;FOLD LIN P2869 Vel=2 m/s CPDAT2869 Tool[1]:marker Base[0] ;%{PE}
;FOLD Parameters ;%{h}
;Params IlfProvider=kukaroboter.basistech.inlineforms.movement.old; Kuka.IsGlobalPoint=False; Kuka.PointName=P2869; Kuka.BlendingEnabled=False; Kuka.MoveDataName=CPDAT1; Kuka.VelocityPath=2; Kuka.CurrentCDSetIndex=0; Kuka.MovementParameterFieldEnabled=True; IlfCommand=LIN
;ENDFOLD
$BWDSTART = FALSE
LDAT_ACT = LCPDAT2869
FDAT_ACT = FP2869
BAS(#CP_PARAMS, 2.0)
SET_CD_PARAMS (0)
LIN XP2869
;ENDFOLD

;FOLD LIN P2870 Vel=2 m/s CPDAT2870 Tool[1]:marker Base[0] ;%{PE}
;FOLD Parameters ;%{h}
;Params IlfProvider=kukaroboter.basistech.inlineforms.movement.old; Kuka.IsGlobalPoint=False; Kuka.PointName=P2870; Kuka.BlendingEnabled=False; Kuka.MoveDataName=CPDAT1; Kuka.VelocityPath=2; Kuka.CurrentCDSetIndex=0; Kuka.MovementParameterFieldEnabled=True; IlfCommand=LIN
;ENDFOLD
$BWDSTART = FALSE
LDAT_ACT = LCPDAT2870
FDAT_ACT = FP2870
BAS(#CP_PARAMS, 2.0)
SET_CD_PARAMS (0)
LIN XP2870
;ENDFOLD

;FOLD LIN P2871 Vel=2 m/s CPDAT2871 Tool[1]:marker Base[0] ;%{PE}
;FOLD Parameters ;%{h}
;Params IlfProvider=kukaroboter.basistech.inlineforms.movement.old; Kuka.IsGlobalPoint=False; Kuka.PointName=P2871; Kuka.BlendingEnabled=False; Kuka.MoveDataName=CPDAT1; Kuka.VelocityPath=2; Kuka.CurrentCDSetIndex=0; Kuka.MovementParameterFieldEnabled=True; IlfCommand=LIN
;ENDFOLD
$BWDSTART = FALSE
LDAT_ACT = LCPDAT2871
FDAT_ACT = FP2871
BAS(#CP_PARAMS, 2.0)
SET_CD_PARAMS (0)
LIN XP2871
;ENDFOLD

;FOLD LIN P2872 Vel=2 m/s CPDAT2872 Tool[1]:marker Base[0] ;%{PE}
;FOLD Parameters ;%{h}
;Params IlfProvider=kukaroboter.basistech.inlineforms.movement.old; Kuka.IsGlobalPoint=False; Kuka.PointName=P2872; Kuka.BlendingEnabled=False; Kuka.MoveDataName=CPDAT1; Kuka.VelocityPath=2; Kuka.CurrentCDSetIndex=0; Kuka.MovementParameterFieldEnabled=True; IlfCommand=LIN
;ENDFOLD
$BWDSTART = FALSE
LDAT_ACT = LCPDAT2872
FDAT_ACT = FP2872
BAS(#CP_PARAMS, 2.0)
SET_CD_PARAMS (0)
LIN XP2872
;ENDFOLD

;FOLD LIN P2873 Vel=2 m/s CPDAT2873 Tool[1]:marker Base[0] ;%{PE}
;FOLD Parameters ;%{h}
;Params IlfProvider=kukaroboter.basistech.inlineforms.movement.old; Kuka.IsGlobalPoint=False; Kuka.PointName=P2873; Kuka.BlendingEnabled=False; Kuka.MoveDataName=CPDAT1; Kuka.VelocityPath=2; Kuka.CurrentCDSetIndex=0; Kuka.MovementParameterFieldEnabled=True; IlfCommand=LIN
;ENDFOLD
$BWDSTART = FALSE
LDAT_ACT = LCPDAT2873
FDAT_ACT = FP2873
BAS(#CP_PARAMS, 2.0)
SET_CD_PARAMS (0)
LIN XP2873
;ENDFOLD

;FOLD LIN P2874 Vel=2 m/s CPDAT2874 Tool[1]:marker Base[0] ;%{PE}
;FOLD Parameters ;%{h}
;Params IlfProvider=kukaroboter.basistech.inlineforms.movement.old; Kuka.IsGlobalPoint=False; Kuka.PointName=P2874; Kuka.BlendingEnabled=False; Kuka.MoveDataName=CPDAT1; Kuka.VelocityPath=2; Kuka.CurrentCDSetIndex=0; Kuka.MovementParameterFieldEnabled=True; IlfCommand=LIN
;ENDFOLD
$BWDSTART = FALSE
LDAT_ACT = LCPDAT2874
FDAT_ACT = FP2874
BAS(#CP_PARAMS, 2.0)
SET_CD_PARAMS (0)
LIN XP2874
;ENDFOLD

;FOLD LIN P2875 Vel=2 m/s CPDAT2875 Tool[1]:marker Base[0] ;%{PE}
;FOLD Parameters ;%{h}
;Params IlfProvider=kukaroboter.basistech.inlineforms.movement.old; Kuka.IsGlobalPoint=False; Kuka.PointName=P2875; Kuka.BlendingEnabled=False; Kuka.MoveDataName=CPDAT1; Kuka.VelocityPath=2; Kuka.CurrentCDSetIndex=0; Kuka.MovementParameterFieldEnabled=True; IlfCommand=LIN
;ENDFOLD
$BWDSTART = FALSE
LDAT_ACT = LCPDAT2875
FDAT_ACT = FP2875
BAS(#CP_PARAMS, 2.0)
SET_CD_PARAMS (0)
LIN XP2875
;ENDFOLD

;FOLD LIN P2876 Vel=2 m/s CPDAT2876 Tool[1]:marker Base[0] ;%{PE}
;FOLD Parameters ;%{h}
;Params IlfProvider=kukaroboter.basistech.inlineforms.movement.old; Kuka.IsGlobalPoint=False; Kuka.PointName=P2876; Kuka.BlendingEnabled=False; Kuka.MoveDataName=CPDAT1; Kuka.VelocityPath=2; Kuka.CurrentCDSetIndex=0; Kuka.MovementParameterFieldEnabled=True; IlfCommand=LIN
;ENDFOLD
$BWDSTART = FALSE
LDAT_ACT = LCPDAT2876
FDAT_ACT = FP2876
BAS(#CP_PARAMS, 2.0)
SET_CD_PARAMS (0)
LIN XP2876
;ENDFOLD

;FOLD LIN P2877 Vel=2 m/s CPDAT2877 Tool[1]:marker Base[0] ;%{PE}
;FOLD Parameters ;%{h}
;Params IlfProvider=kukaroboter.basistech.inlineforms.movement.old; Kuka.IsGlobalPoint=False; Kuka.PointName=P2877; Kuka.BlendingEnabled=False; Kuka.MoveDataName=CPDAT1; Kuka.VelocityPath=2; Kuka.CurrentCDSetIndex=0; Kuka.MovementParameterFieldEnabled=True; IlfCommand=LIN
;ENDFOLD
$BWDSTART = FALSE
LDAT_ACT = LCPDAT2877
FDAT_ACT = FP2877
BAS(#CP_PARAMS, 2.0)
SET_CD_PARAMS (0)
LIN XP2877
;ENDFOLD

;FOLD LIN P2878 Vel=2 m/s CPDAT2878 Tool[1]:marker Base[0] ;%{PE}
;FOLD Parameters ;%{h}
;Params IlfProvider=kukaroboter.basistech.inlineforms.movement.old; Kuka.IsGlobalPoint=False; Kuka.PointName=P2878; Kuka.BlendingEnabled=False; Kuka.MoveDataName=CPDAT1; Kuka.VelocityPath=2; Kuka.CurrentCDSetIndex=0; Kuka.MovementParameterFieldEnabled=True; IlfCommand=LIN
;ENDFOLD
$BWDSTART = FALSE
LDAT_ACT = LCPDAT2878
FDAT_ACT = FP2878
BAS(#CP_PARAMS, 2.0)
SET_CD_PARAMS (0)
LIN XP2878
;ENDFOLD

;FOLD LIN P2879 Vel=2 m/s CPDAT2879 Tool[1]:marker Base[0] ;%{PE}
;FOLD Parameters ;%{h}
;Params IlfProvider=kukaroboter.basistech.inlineforms.movement.old; Kuka.IsGlobalPoint=False; Kuka.PointName=P2879; Kuka.BlendingEnabled=False; Kuka.MoveDataName=CPDAT1; Kuka.VelocityPath=2; Kuka.CurrentCDSetIndex=0; Kuka.MovementParameterFieldEnabled=True; IlfCommand=LIN
;ENDFOLD
$BWDSTART = FALSE
LDAT_ACT = LCPDAT2879
FDAT_ACT = FP2879
BAS(#CP_PARAMS, 2.0)
SET_CD_PARAMS (0)
LIN XP2879
;ENDFOLD

;FOLD LIN P2880 Vel=2 m/s CPDAT2880 Tool[1]:marker Base[0] ;%{PE}
;FOLD Parameters ;%{h}
;Params IlfProvider=kukaroboter.basistech.inlineforms.movement.old; Kuka.IsGlobalPoint=False; Kuka.PointName=P2880; Kuka.BlendingEnabled=False; Kuka.MoveDataName=CPDAT1; Kuka.VelocityPath=2; Kuka.CurrentCDSetIndex=0; Kuka.MovementParameterFieldEnabled=True; IlfCommand=LIN
;ENDFOLD
$BWDSTART = FALSE
LDAT_ACT = LCPDAT2880
FDAT_ACT = FP2880
BAS(#CP_PARAMS, 2.0)
SET_CD_PARAMS (0)
LIN XP2880
;ENDFOLD

;FOLD LIN P2881 Vel=2 m/s CPDAT2881 Tool[1]:marker Base[0] ;%{PE}
;FOLD Parameters ;%{h}
;Params IlfProvider=kukaroboter.basistech.inlineforms.movement.old; Kuka.IsGlobalPoint=False; Kuka.PointName=P2881; Kuka.BlendingEnabled=False; Kuka.MoveDataName=CPDAT1; Kuka.VelocityPath=2; Kuka.CurrentCDSetIndex=0; Kuka.MovementParameterFieldEnabled=True; IlfCommand=LIN
;ENDFOLD
$BWDSTART = FALSE
LDAT_ACT = LCPDAT2881
FDAT_ACT = FP2881
BAS(#CP_PARAMS, 2.0)
SET_CD_PARAMS (0)
LIN XP2881
;ENDFOLD

;FOLD LIN P2882 Vel=2 m/s CPDAT2882 Tool[1]:marker Base[0] ;%{PE}
;FOLD Parameters ;%{h}
;Params IlfProvider=kukaroboter.basistech.inlineforms.movement.old; Kuka.IsGlobalPoint=False; Kuka.PointName=P2882; Kuka.BlendingEnabled=False; Kuka.MoveDataName=CPDAT1; Kuka.VelocityPath=2; Kuka.CurrentCDSetIndex=0; Kuka.MovementParameterFieldEnabled=True; IlfCommand=LIN
;ENDFOLD
$BWDSTART = FALSE
LDAT_ACT = LCPDAT2882
FDAT_ACT = FP2882
BAS(#CP_PARAMS, 2.0)
SET_CD_PARAMS (0)
LIN XP2882
;ENDFOLD

;FOLD LIN P2883 Vel=2 m/s CPDAT2883 Tool[1]:marker Base[0] ;%{PE}
;FOLD Parameters ;%{h}
;Params IlfProvider=kukaroboter.basistech.inlineforms.movement.old; Kuka.IsGlobalPoint=False; Kuka.PointName=P2883; Kuka.BlendingEnabled=False; Kuka.MoveDataName=CPDAT1; Kuka.VelocityPath=2; Kuka.CurrentCDSetIndex=0; Kuka.MovementParameterFieldEnabled=True; IlfCommand=LIN
;ENDFOLD
$BWDSTART = FALSE
LDAT_ACT = LCPDAT2883
FDAT_ACT = FP2883
BAS(#CP_PARAMS, 2.0)
SET_CD_PARAMS (0)
LIN XP2883
;ENDFOLD

;FOLD LIN P2884 Vel=2 m/s CPDAT2884 Tool[1]:marker Base[0] ;%{PE}
;FOLD Parameters ;%{h}
;Params IlfProvider=kukaroboter.basistech.inlineforms.movement.old; Kuka.IsGlobalPoint=False; Kuka.PointName=P2884; Kuka.BlendingEnabled=False; Kuka.MoveDataName=CPDAT1; Kuka.VelocityPath=2; Kuka.CurrentCDSetIndex=0; Kuka.MovementParameterFieldEnabled=True; IlfCommand=LIN
;ENDFOLD
$BWDSTART = FALSE
LDAT_ACT = LCPDAT2884
FDAT_ACT = FP2884
BAS(#CP_PARAMS, 2.0)
SET_CD_PARAMS (0)
LIN XP2884
;ENDFOLD

;FOLD LIN P2885 Vel=2 m/s CPDAT2885 Tool[1]:marker Base[0] ;%{PE}
;FOLD Parameters ;%{h}
;Params IlfProvider=kukaroboter.basistech.inlineforms.movement.old; Kuka.IsGlobalPoint=False; Kuka.PointName=P2885; Kuka.BlendingEnabled=False; Kuka.MoveDataName=CPDAT1; Kuka.VelocityPath=2; Kuka.CurrentCDSetIndex=0; Kuka.MovementParameterFieldEnabled=True; IlfCommand=LIN
;ENDFOLD
$BWDSTART = FALSE
LDAT_ACT = LCPDAT2885
FDAT_ACT = FP2885
BAS(#CP_PARAMS, 2.0)
SET_CD_PARAMS (0)
LIN XP2885
;ENDFOLD

;FOLD LIN P2886 Vel=2 m/s CPDAT2886 Tool[1]:marker Base[0] ;%{PE}
;FOLD Parameters ;%{h}
;Params IlfProvider=kukaroboter.basistech.inlineforms.movement.old; Kuka.IsGlobalPoint=False; Kuka.PointName=P2886; Kuka.BlendingEnabled=False; Kuka.MoveDataName=CPDAT1; Kuka.VelocityPath=2; Kuka.CurrentCDSetIndex=0; Kuka.MovementParameterFieldEnabled=True; IlfCommand=LIN
;ENDFOLD
$BWDSTART = FALSE
LDAT_ACT = LCPDAT2886
FDAT_ACT = FP2886
BAS(#CP_PARAMS, 2.0)
SET_CD_PARAMS (0)
LIN XP2886
;ENDFOLD

;FOLD LIN P2887 Vel=2 m/s CPDAT2887 Tool[1]:marker Base[0] ;%{PE}
;FOLD Parameters ;%{h}
;Params IlfProvider=kukaroboter.basistech.inlineforms.movement.old; Kuka.IsGlobalPoint=False; Kuka.PointName=P2887; Kuka.BlendingEnabled=False; Kuka.MoveDataName=CPDAT1; Kuka.VelocityPath=2; Kuka.CurrentCDSetIndex=0; Kuka.MovementParameterFieldEnabled=True; IlfCommand=LIN
;ENDFOLD
$BWDSTART = FALSE
LDAT_ACT = LCPDAT2887
FDAT_ACT = FP2887
BAS(#CP_PARAMS, 2.0)
SET_CD_PARAMS (0)
LIN XP2887
;ENDFOLD

;FOLD LIN P2888 Vel=2 m/s CPDAT2888 Tool[1]:marker Base[0] ;%{PE}
;FOLD Parameters ;%{h}
;Params IlfProvider=kukaroboter.basistech.inlineforms.movement.old; Kuka.IsGlobalPoint=False; Kuka.PointName=P2888; Kuka.BlendingEnabled=False; Kuka.MoveDataName=CPDAT1; Kuka.VelocityPath=2; Kuka.CurrentCDSetIndex=0; Kuka.MovementParameterFieldEnabled=True; IlfCommand=LIN
;ENDFOLD
$BWDSTART = FALSE
LDAT_ACT = LCPDAT2888
FDAT_ACT = FP2888
BAS(#CP_PARAMS, 2.0)
SET_CD_PARAMS (0)
LIN XP2888
;ENDFOLD

;FOLD LIN P2889 Vel=2 m/s CPDAT2889 Tool[1]:marker Base[0] ;%{PE}
;FOLD Parameters ;%{h}
;Params IlfProvider=kukaroboter.basistech.inlineforms.movement.old; Kuka.IsGlobalPoint=False; Kuka.PointName=P2889; Kuka.BlendingEnabled=False; Kuka.MoveDataName=CPDAT1; Kuka.VelocityPath=2; Kuka.CurrentCDSetIndex=0; Kuka.MovementParameterFieldEnabled=True; IlfCommand=LIN
;ENDFOLD
$BWDSTART = FALSE
LDAT_ACT = LCPDAT2889
FDAT_ACT = FP2889
BAS(#CP_PARAMS, 2.0)
SET_CD_PARAMS (0)
LIN XP2889
;ENDFOLD

;FOLD LIN P2890 Vel=2 m/s CPDAT2890 Tool[1]:marker Base[0] ;%{PE}
;FOLD Parameters ;%{h}
;Params IlfProvider=kukaroboter.basistech.inlineforms.movement.old; Kuka.IsGlobalPoint=False; Kuka.PointName=P2890; Kuka.BlendingEnabled=False; Kuka.MoveDataName=CPDAT1; Kuka.VelocityPath=2; Kuka.CurrentCDSetIndex=0; Kuka.MovementParameterFieldEnabled=True; IlfCommand=LIN
;ENDFOLD
$BWDSTART = FALSE
LDAT_ACT = LCPDAT2890
FDAT_ACT = FP2890
BAS(#CP_PARAMS, 2.0)
SET_CD_PARAMS (0)
LIN XP2890
;ENDFOLD

;FOLD LIN P2891 Vel=2 m/s CPDAT2891 Tool[1]:marker Base[0] ;%{PE}
;FOLD Parameters ;%{h}
;Params IlfProvider=kukaroboter.basistech.inlineforms.movement.old; Kuka.IsGlobalPoint=False; Kuka.PointName=P2891; Kuka.BlendingEnabled=False; Kuka.MoveDataName=CPDAT1; Kuka.VelocityPath=2; Kuka.CurrentCDSetIndex=0; Kuka.MovementParameterFieldEnabled=True; IlfCommand=LIN
;ENDFOLD
$BWDSTART = FALSE
LDAT_ACT = LCPDAT2891
FDAT_ACT = FP2891
BAS(#CP_PARAMS, 2.0)
SET_CD_PARAMS (0)
LIN XP2891
;ENDFOLD

;FOLD LIN P2892 Vel=2 m/s CPDAT2892 Tool[1]:marker Base[0] ;%{PE}
;FOLD Parameters ;%{h}
;Params IlfProvider=kukaroboter.basistech.inlineforms.movement.old; Kuka.IsGlobalPoint=False; Kuka.PointName=P2892; Kuka.BlendingEnabled=False; Kuka.MoveDataName=CPDAT1; Kuka.VelocityPath=2; Kuka.CurrentCDSetIndex=0; Kuka.MovementParameterFieldEnabled=True; IlfCommand=LIN
;ENDFOLD
$BWDSTART = FALSE
LDAT_ACT = LCPDAT2892
FDAT_ACT = FP2892
BAS(#CP_PARAMS, 2.0)
SET_CD_PARAMS (0)
LIN XP2892
;ENDFOLD

;FOLD LIN P2893 Vel=2 m/s CPDAT2893 Tool[1]:marker Base[0] ;%{PE}
;FOLD Parameters ;%{h}
;Params IlfProvider=kukaroboter.basistech.inlineforms.movement.old; Kuka.IsGlobalPoint=False; Kuka.PointName=P2893; Kuka.BlendingEnabled=False; Kuka.MoveDataName=CPDAT1; Kuka.VelocityPath=2; Kuka.CurrentCDSetIndex=0; Kuka.MovementParameterFieldEnabled=True; IlfCommand=LIN
;ENDFOLD
$BWDSTART = FALSE
LDAT_ACT = LCPDAT2893
FDAT_ACT = FP2893
BAS(#CP_PARAMS, 2.0)
SET_CD_PARAMS (0)
LIN XP2893
;ENDFOLD

;FOLD LIN P2894 Vel=2 m/s CPDAT2894 Tool[1]:marker Base[0] ;%{PE}
;FOLD Parameters ;%{h}
;Params IlfProvider=kukaroboter.basistech.inlineforms.movement.old; Kuka.IsGlobalPoint=False; Kuka.PointName=P2894; Kuka.BlendingEnabled=False; Kuka.MoveDataName=CPDAT1; Kuka.VelocityPath=2; Kuka.CurrentCDSetIndex=0; Kuka.MovementParameterFieldEnabled=True; IlfCommand=LIN
;ENDFOLD
$BWDSTART = FALSE
LDAT_ACT = LCPDAT2894
FDAT_ACT = FP2894
BAS(#CP_PARAMS, 2.0)
SET_CD_PARAMS (0)
LIN XP2894
;ENDFOLD

;FOLD LIN P2895 Vel=2 m/s CPDAT2895 Tool[1]:marker Base[0] ;%{PE}
;FOLD Parameters ;%{h}
;Params IlfProvider=kukaroboter.basistech.inlineforms.movement.old; Kuka.IsGlobalPoint=False; Kuka.PointName=P2895; Kuka.BlendingEnabled=False; Kuka.MoveDataName=CPDAT1; Kuka.VelocityPath=2; Kuka.CurrentCDSetIndex=0; Kuka.MovementParameterFieldEnabled=True; IlfCommand=LIN
;ENDFOLD
$BWDSTART = FALSE
LDAT_ACT = LCPDAT2895
FDAT_ACT = FP2895
BAS(#CP_PARAMS, 2.0)
SET_CD_PARAMS (0)
LIN XP2895
;ENDFOLD

;FOLD LIN P2896 Vel=2 m/s CPDAT2896 Tool[1]:marker Base[0] ;%{PE}
;FOLD Parameters ;%{h}
;Params IlfProvider=kukaroboter.basistech.inlineforms.movement.old; Kuka.IsGlobalPoint=False; Kuka.PointName=P2896; Kuka.BlendingEnabled=False; Kuka.MoveDataName=CPDAT1; Kuka.VelocityPath=2; Kuka.CurrentCDSetIndex=0; Kuka.MovementParameterFieldEnabled=True; IlfCommand=LIN
;ENDFOLD
$BWDSTART = FALSE
LDAT_ACT = LCPDAT2896
FDAT_ACT = FP2896
BAS(#CP_PARAMS, 2.0)
SET_CD_PARAMS (0)
LIN XP2896
;ENDFOLD

;FOLD LIN P2897 Vel=2 m/s CPDAT2897 Tool[1]:marker Base[0] ;%{PE}
;FOLD Parameters ;%{h}
;Params IlfProvider=kukaroboter.basistech.inlineforms.movement.old; Kuka.IsGlobalPoint=False; Kuka.PointName=P2897; Kuka.BlendingEnabled=False; Kuka.MoveDataName=CPDAT1; Kuka.VelocityPath=2; Kuka.CurrentCDSetIndex=0; Kuka.MovementParameterFieldEnabled=True; IlfCommand=LIN
;ENDFOLD
$BWDSTART = FALSE
LDAT_ACT = LCPDAT2897
FDAT_ACT = FP2897
BAS(#CP_PARAMS, 2.0)
SET_CD_PARAMS (0)
LIN XP2897
;ENDFOLD

;FOLD LIN P2898 Vel=2 m/s CPDAT2898 Tool[1]:marker Base[0] ;%{PE}
;FOLD Parameters ;%{h}
;Params IlfProvider=kukaroboter.basistech.inlineforms.movement.old; Kuka.IsGlobalPoint=False; Kuka.PointName=P2898; Kuka.BlendingEnabled=False; Kuka.MoveDataName=CPDAT1; Kuka.VelocityPath=2; Kuka.CurrentCDSetIndex=0; Kuka.MovementParameterFieldEnabled=True; IlfCommand=LIN
;ENDFOLD
$BWDSTART = FALSE
LDAT_ACT = LCPDAT2898
FDAT_ACT = FP2898
BAS(#CP_PARAMS, 2.0)
SET_CD_PARAMS (0)
LIN XP2898
;ENDFOLD

;FOLD LIN P2899 Vel=2 m/s CPDAT2899 Tool[1]:marker Base[0] ;%{PE}
;FOLD Parameters ;%{h}
;Params IlfProvider=kukaroboter.basistech.inlineforms.movement.old; Kuka.IsGlobalPoint=False; Kuka.PointName=P2899; Kuka.BlendingEnabled=False; Kuka.MoveDataName=CPDAT1; Kuka.VelocityPath=2; Kuka.CurrentCDSetIndex=0; Kuka.MovementParameterFieldEnabled=True; IlfCommand=LIN
;ENDFOLD
$BWDSTART = FALSE
LDAT_ACT = LCPDAT2899
FDAT_ACT = FP2899
BAS(#CP_PARAMS, 2.0)
SET_CD_PARAMS (0)
LIN XP2899
;ENDFOLD

;FOLD LIN P2900 Vel=2 m/s CPDAT2900 Tool[1]:marker Base[0] ;%{PE}
;FOLD Parameters ;%{h}
;Params IlfProvider=kukaroboter.basistech.inlineforms.movement.old; Kuka.IsGlobalPoint=False; Kuka.PointName=P2900; Kuka.BlendingEnabled=False; Kuka.MoveDataName=CPDAT1; Kuka.VelocityPath=2; Kuka.CurrentCDSetIndex=0; Kuka.MovementParameterFieldEnabled=True; IlfCommand=LIN
;ENDFOLD
$BWDSTART = FALSE
LDAT_ACT = LCPDAT2900
FDAT_ACT = FP2900
BAS(#CP_PARAMS, 2.0)
SET_CD_PARAMS (0)
LIN XP2900
;ENDFOLD

;FOLD LIN P2901 Vel=2 m/s CPDAT2901 Tool[1]:marker Base[0] ;%{PE}
;FOLD Parameters ;%{h}
;Params IlfProvider=kukaroboter.basistech.inlineforms.movement.old; Kuka.IsGlobalPoint=False; Kuka.PointName=P2901; Kuka.BlendingEnabled=False; Kuka.MoveDataName=CPDAT1; Kuka.VelocityPath=2; Kuka.CurrentCDSetIndex=0; Kuka.MovementParameterFieldEnabled=True; IlfCommand=LIN
;ENDFOLD
$BWDSTART = FALSE
LDAT_ACT = LCPDAT2901
FDAT_ACT = FP2901
BAS(#CP_PARAMS, 2.0)
SET_CD_PARAMS (0)
LIN XP2901
;ENDFOLD

;FOLD LIN P2902 Vel=2 m/s CPDAT2902 Tool[1]:marker Base[0] ;%{PE}
;FOLD Parameters ;%{h}
;Params IlfProvider=kukaroboter.basistech.inlineforms.movement.old; Kuka.IsGlobalPoint=False; Kuka.PointName=P2902; Kuka.BlendingEnabled=False; Kuka.MoveDataName=CPDAT1; Kuka.VelocityPath=2; Kuka.CurrentCDSetIndex=0; Kuka.MovementParameterFieldEnabled=True; IlfCommand=LIN
;ENDFOLD
$BWDSTART = FALSE
LDAT_ACT = LCPDAT2902
FDAT_ACT = FP2902
BAS(#CP_PARAMS, 2.0)
SET_CD_PARAMS (0)
LIN XP2902
;ENDFOLD

;FOLD LIN P2903 Vel=2 m/s CPDAT2903 Tool[1]:marker Base[0] ;%{PE}
;FOLD Parameters ;%{h}
;Params IlfProvider=kukaroboter.basistech.inlineforms.movement.old; Kuka.IsGlobalPoint=False; Kuka.PointName=P2903; Kuka.BlendingEnabled=False; Kuka.MoveDataName=CPDAT1; Kuka.VelocityPath=2; Kuka.CurrentCDSetIndex=0; Kuka.MovementParameterFieldEnabled=True; IlfCommand=LIN
;ENDFOLD
$BWDSTART = FALSE
LDAT_ACT = LCPDAT2903
FDAT_ACT = FP2903
BAS(#CP_PARAMS, 2.0)
SET_CD_PARAMS (0)
LIN XP2903
;ENDFOLD

;FOLD LIN P2904 Vel=2 m/s CPDAT2904 Tool[1]:marker Base[0] ;%{PE}
;FOLD Parameters ;%{h}
;Params IlfProvider=kukaroboter.basistech.inlineforms.movement.old; Kuka.IsGlobalPoint=False; Kuka.PointName=P2904; Kuka.BlendingEnabled=False; Kuka.MoveDataName=CPDAT1; Kuka.VelocityPath=2; Kuka.CurrentCDSetIndex=0; Kuka.MovementParameterFieldEnabled=True; IlfCommand=LIN
;ENDFOLD
$BWDSTART = FALSE
LDAT_ACT = LCPDAT2904
FDAT_ACT = FP2904
BAS(#CP_PARAMS, 2.0)
SET_CD_PARAMS (0)
LIN XP2904
;ENDFOLD

;FOLD LIN P2905 Vel=2 m/s CPDAT2905 Tool[1]:marker Base[0] ;%{PE}
;FOLD Parameters ;%{h}
;Params IlfProvider=kukaroboter.basistech.inlineforms.movement.old; Kuka.IsGlobalPoint=False; Kuka.PointName=P2905; Kuka.BlendingEnabled=False; Kuka.MoveDataName=CPDAT1; Kuka.VelocityPath=2; Kuka.CurrentCDSetIndex=0; Kuka.MovementParameterFieldEnabled=True; IlfCommand=LIN
;ENDFOLD
$BWDSTART = FALSE
LDAT_ACT = LCPDAT2905
FDAT_ACT = FP2905
BAS(#CP_PARAMS, 2.0)
SET_CD_PARAMS (0)
LIN XP2905
;ENDFOLD

;FOLD LIN P2906 Vel=2 m/s CPDAT2906 Tool[1]:marker Base[0] ;%{PE}
;FOLD Parameters ;%{h}
;Params IlfProvider=kukaroboter.basistech.inlineforms.movement.old; Kuka.IsGlobalPoint=False; Kuka.PointName=P2906; Kuka.BlendingEnabled=False; Kuka.MoveDataName=CPDAT1; Kuka.VelocityPath=2; Kuka.CurrentCDSetIndex=0; Kuka.MovementParameterFieldEnabled=True; IlfCommand=LIN
;ENDFOLD
$BWDSTART = FALSE
LDAT_ACT = LCPDAT2906
FDAT_ACT = FP2906
BAS(#CP_PARAMS, 2.0)
SET_CD_PARAMS (0)
LIN XP2906
;ENDFOLD

;FOLD LIN P2907 Vel=2 m/s CPDAT2907 Tool[1]:marker Base[0] ;%{PE}
;FOLD Parameters ;%{h}
;Params IlfProvider=kukaroboter.basistech.inlineforms.movement.old; Kuka.IsGlobalPoint=False; Kuka.PointName=P2907; Kuka.BlendingEnabled=False; Kuka.MoveDataName=CPDAT1; Kuka.VelocityPath=2; Kuka.CurrentCDSetIndex=0; Kuka.MovementParameterFieldEnabled=True; IlfCommand=LIN
;ENDFOLD
$BWDSTART = FALSE
LDAT_ACT = LCPDAT2907
FDAT_ACT = FP2907
BAS(#CP_PARAMS, 2.0)
SET_CD_PARAMS (0)
LIN XP2907
;ENDFOLD

;FOLD LIN P2908 Vel=2 m/s CPDAT2908 Tool[1]:marker Base[0] ;%{PE}
;FOLD Parameters ;%{h}
;Params IlfProvider=kukaroboter.basistech.inlineforms.movement.old; Kuka.IsGlobalPoint=False; Kuka.PointName=P2908; Kuka.BlendingEnabled=False; Kuka.MoveDataName=CPDAT1; Kuka.VelocityPath=2; Kuka.CurrentCDSetIndex=0; Kuka.MovementParameterFieldEnabled=True; IlfCommand=LIN
;ENDFOLD
$BWDSTART = FALSE
LDAT_ACT = LCPDAT2908
FDAT_ACT = FP2908
BAS(#CP_PARAMS, 2.0)
SET_CD_PARAMS (0)
LIN XP2908
;ENDFOLD

;FOLD LIN P2909 Vel=2 m/s CPDAT2909 Tool[1]:marker Base[0] ;%{PE}
;FOLD Parameters ;%{h}
;Params IlfProvider=kukaroboter.basistech.inlineforms.movement.old; Kuka.IsGlobalPoint=False; Kuka.PointName=P2909; Kuka.BlendingEnabled=False; Kuka.MoveDataName=CPDAT1; Kuka.VelocityPath=2; Kuka.CurrentCDSetIndex=0; Kuka.MovementParameterFieldEnabled=True; IlfCommand=LIN
;ENDFOLD
$BWDSTART = FALSE
LDAT_ACT = LCPDAT2909
FDAT_ACT = FP2909
BAS(#CP_PARAMS, 2.0)
SET_CD_PARAMS (0)
LIN XP2909
;ENDFOLD

;FOLD LIN P2910 Vel=2 m/s CPDAT2910 Tool[1]:marker Base[0] ;%{PE}
;FOLD Parameters ;%{h}
;Params IlfProvider=kukaroboter.basistech.inlineforms.movement.old; Kuka.IsGlobalPoint=False; Kuka.PointName=P2910; Kuka.BlendingEnabled=False; Kuka.MoveDataName=CPDAT1; Kuka.VelocityPath=2; Kuka.CurrentCDSetIndex=0; Kuka.MovementParameterFieldEnabled=True; IlfCommand=LIN
;ENDFOLD
$BWDSTART = FALSE
LDAT_ACT = LCPDAT2910
FDAT_ACT = FP2910
BAS(#CP_PARAMS, 2.0)
SET_CD_PARAMS (0)
LIN XP2910
;ENDFOLD

;FOLD LIN P2911 Vel=2 m/s CPDAT2911 Tool[1]:marker Base[0] ;%{PE}
;FOLD Parameters ;%{h}
;Params IlfProvider=kukaroboter.basistech.inlineforms.movement.old; Kuka.IsGlobalPoint=False; Kuka.PointName=P2911; Kuka.BlendingEnabled=False; Kuka.MoveDataName=CPDAT1; Kuka.VelocityPath=2; Kuka.CurrentCDSetIndex=0; Kuka.MovementParameterFieldEnabled=True; IlfCommand=LIN
;ENDFOLD
$BWDSTART = FALSE
LDAT_ACT = LCPDAT2911
FDAT_ACT = FP2911
BAS(#CP_PARAMS, 2.0)
SET_CD_PARAMS (0)
LIN XP2911
;ENDFOLD

;FOLD LIN P2912 Vel=2 m/s CPDAT2912 Tool[1]:marker Base[0] ;%{PE}
;FOLD Parameters ;%{h}
;Params IlfProvider=kukaroboter.basistech.inlineforms.movement.old; Kuka.IsGlobalPoint=False; Kuka.PointName=P2912; Kuka.BlendingEnabled=False; Kuka.MoveDataName=CPDAT1; Kuka.VelocityPath=2; Kuka.CurrentCDSetIndex=0; Kuka.MovementParameterFieldEnabled=True; IlfCommand=LIN
;ENDFOLD
$BWDSTART = FALSE
LDAT_ACT = LCPDAT2912
FDAT_ACT = FP2912
BAS(#CP_PARAMS, 2.0)
SET_CD_PARAMS (0)
LIN XP2912
;ENDFOLD

;FOLD LIN P2913 Vel=2 m/s CPDAT2913 Tool[1]:marker Base[0] ;%{PE}
;FOLD Parameters ;%{h}
;Params IlfProvider=kukaroboter.basistech.inlineforms.movement.old; Kuka.IsGlobalPoint=False; Kuka.PointName=P2913; Kuka.BlendingEnabled=False; Kuka.MoveDataName=CPDAT1; Kuka.VelocityPath=2; Kuka.CurrentCDSetIndex=0; Kuka.MovementParameterFieldEnabled=True; IlfCommand=LIN
;ENDFOLD
$BWDSTART = FALSE
LDAT_ACT = LCPDAT2913
FDAT_ACT = FP2913
BAS(#CP_PARAMS, 2.0)
SET_CD_PARAMS (0)
LIN XP2913
;ENDFOLD

;FOLD LIN P2914 Vel=2 m/s CPDAT2914 Tool[1]:marker Base[0] ;%{PE}
;FOLD Parameters ;%{h}
;Params IlfProvider=kukaroboter.basistech.inlineforms.movement.old; Kuka.IsGlobalPoint=False; Kuka.PointName=P2914; Kuka.BlendingEnabled=False; Kuka.MoveDataName=CPDAT1; Kuka.VelocityPath=2; Kuka.CurrentCDSetIndex=0; Kuka.MovementParameterFieldEnabled=True; IlfCommand=LIN
;ENDFOLD
$BWDSTART = FALSE
LDAT_ACT = LCPDAT2914
FDAT_ACT = FP2914
BAS(#CP_PARAMS, 2.0)
SET_CD_PARAMS (0)
LIN XP2914
;ENDFOLD

;FOLD LIN P2915 Vel=2 m/s CPDAT2915 Tool[1]:marker Base[0] ;%{PE}
;FOLD Parameters ;%{h}
;Params IlfProvider=kukaroboter.basistech.inlineforms.movement.old; Kuka.IsGlobalPoint=False; Kuka.PointName=P2915; Kuka.BlendingEnabled=False; Kuka.MoveDataName=CPDAT1; Kuka.VelocityPath=2; Kuka.CurrentCDSetIndex=0; Kuka.MovementParameterFieldEnabled=True; IlfCommand=LIN
;ENDFOLD
$BWDSTART = FALSE
LDAT_ACT = LCPDAT2915
FDAT_ACT = FP2915
BAS(#CP_PARAMS, 2.0)
SET_CD_PARAMS (0)
LIN XP2915
;ENDFOLD

;FOLD LIN P2916 Vel=2 m/s CPDAT2916 Tool[1]:marker Base[0] ;%{PE}
;FOLD Parameters ;%{h}
;Params IlfProvider=kukaroboter.basistech.inlineforms.movement.old; Kuka.IsGlobalPoint=False; Kuka.PointName=P2916; Kuka.BlendingEnabled=False; Kuka.MoveDataName=CPDAT1; Kuka.VelocityPath=2; Kuka.CurrentCDSetIndex=0; Kuka.MovementParameterFieldEnabled=True; IlfCommand=LIN
;ENDFOLD
$BWDSTART = FALSE
LDAT_ACT = LCPDAT2916
FDAT_ACT = FP2916
BAS(#CP_PARAMS, 2.0)
SET_CD_PARAMS (0)
LIN XP2916
;ENDFOLD

;FOLD LIN P2917 Vel=2 m/s CPDAT2917 Tool[1]:marker Base[0] ;%{PE}
;FOLD Parameters ;%{h}
;Params IlfProvider=kukaroboter.basistech.inlineforms.movement.old; Kuka.IsGlobalPoint=False; Kuka.PointName=P2917; Kuka.BlendingEnabled=False; Kuka.MoveDataName=CPDAT1; Kuka.VelocityPath=2; Kuka.CurrentCDSetIndex=0; Kuka.MovementParameterFieldEnabled=True; IlfCommand=LIN
;ENDFOLD
$BWDSTART = FALSE
LDAT_ACT = LCPDAT2917
FDAT_ACT = FP2917
BAS(#CP_PARAMS, 2.0)
SET_CD_PARAMS (0)
LIN XP2917
;ENDFOLD

;FOLD LIN P2918 Vel=2 m/s CPDAT2918 Tool[1]:marker Base[0] ;%{PE}
;FOLD Parameters ;%{h}
;Params IlfProvider=kukaroboter.basistech.inlineforms.movement.old; Kuka.IsGlobalPoint=False; Kuka.PointName=P2918; Kuka.BlendingEnabled=False; Kuka.MoveDataName=CPDAT1; Kuka.VelocityPath=2; Kuka.CurrentCDSetIndex=0; Kuka.MovementParameterFieldEnabled=True; IlfCommand=LIN
;ENDFOLD
$BWDSTART = FALSE
LDAT_ACT = LCPDAT2918
FDAT_ACT = FP2918
BAS(#CP_PARAMS, 2.0)
SET_CD_PARAMS (0)
LIN XP2918
;ENDFOLD

;FOLD LIN P2919 Vel=2 m/s CPDAT2919 Tool[1]:marker Base[0] ;%{PE}
;FOLD Parameters ;%{h}
;Params IlfProvider=kukaroboter.basistech.inlineforms.movement.old; Kuka.IsGlobalPoint=False; Kuka.PointName=P2919; Kuka.BlendingEnabled=False; Kuka.MoveDataName=CPDAT1; Kuka.VelocityPath=2; Kuka.CurrentCDSetIndex=0; Kuka.MovementParameterFieldEnabled=True; IlfCommand=LIN
;ENDFOLD
$BWDSTART = FALSE
LDAT_ACT = LCPDAT2919
FDAT_ACT = FP2919
BAS(#CP_PARAMS, 2.0)
SET_CD_PARAMS (0)
LIN XP2919
;ENDFOLD

;FOLD LIN P2920 Vel=2 m/s CPDAT2920 Tool[1]:marker Base[0] ;%{PE}
;FOLD Parameters ;%{h}
;Params IlfProvider=kukaroboter.basistech.inlineforms.movement.old; Kuka.IsGlobalPoint=False; Kuka.PointName=P2920; Kuka.BlendingEnabled=False; Kuka.MoveDataName=CPDAT1; Kuka.VelocityPath=2; Kuka.CurrentCDSetIndex=0; Kuka.MovementParameterFieldEnabled=True; IlfCommand=LIN
;ENDFOLD
$BWDSTART = FALSE
LDAT_ACT = LCPDAT2920
FDAT_ACT = FP2920
BAS(#CP_PARAMS, 2.0)
SET_CD_PARAMS (0)
LIN XP2920
;ENDFOLD

;FOLD LIN P2921 Vel=2 m/s CPDAT2921 Tool[1]:marker Base[0] ;%{PE}
;FOLD Parameters ;%{h}
;Params IlfProvider=kukaroboter.basistech.inlineforms.movement.old; Kuka.IsGlobalPoint=False; Kuka.PointName=P2921; Kuka.BlendingEnabled=False; Kuka.MoveDataName=CPDAT1; Kuka.VelocityPath=2; Kuka.CurrentCDSetIndex=0; Kuka.MovementParameterFieldEnabled=True; IlfCommand=LIN
;ENDFOLD
$BWDSTART = FALSE
LDAT_ACT = LCPDAT2921
FDAT_ACT = FP2921
BAS(#CP_PARAMS, 2.0)
SET_CD_PARAMS (0)
LIN XP2921
;ENDFOLD

;FOLD LIN P2922 Vel=2 m/s CPDAT2922 Tool[1]:marker Base[0] ;%{PE}
;FOLD Parameters ;%{h}
;Params IlfProvider=kukaroboter.basistech.inlineforms.movement.old; Kuka.IsGlobalPoint=False; Kuka.PointName=P2922; Kuka.BlendingEnabled=False; Kuka.MoveDataName=CPDAT1; Kuka.VelocityPath=2; Kuka.CurrentCDSetIndex=0; Kuka.MovementParameterFieldEnabled=True; IlfCommand=LIN
;ENDFOLD
$BWDSTART = FALSE
LDAT_ACT = LCPDAT2922
FDAT_ACT = FP2922
BAS(#CP_PARAMS, 2.0)
SET_CD_PARAMS (0)
LIN XP2922
;ENDFOLD

;FOLD LIN P2923 Vel=2 m/s CPDAT2923 Tool[1]:marker Base[0] ;%{PE}
;FOLD Parameters ;%{h}
;Params IlfProvider=kukaroboter.basistech.inlineforms.movement.old; Kuka.IsGlobalPoint=False; Kuka.PointName=P2923; Kuka.BlendingEnabled=False; Kuka.MoveDataName=CPDAT1; Kuka.VelocityPath=2; Kuka.CurrentCDSetIndex=0; Kuka.MovementParameterFieldEnabled=True; IlfCommand=LIN
;ENDFOLD
$BWDSTART = FALSE
LDAT_ACT = LCPDAT2923
FDAT_ACT = FP2923
BAS(#CP_PARAMS, 2.0)
SET_CD_PARAMS (0)
LIN XP2923
;ENDFOLD

;FOLD LIN P2924 Vel=2 m/s CPDAT2924 Tool[1]:marker Base[0] ;%{PE}
;FOLD Parameters ;%{h}
;Params IlfProvider=kukaroboter.basistech.inlineforms.movement.old; Kuka.IsGlobalPoint=False; Kuka.PointName=P2924; Kuka.BlendingEnabled=False; Kuka.MoveDataName=CPDAT1; Kuka.VelocityPath=2; Kuka.CurrentCDSetIndex=0; Kuka.MovementParameterFieldEnabled=True; IlfCommand=LIN
;ENDFOLD
$BWDSTART = FALSE
LDAT_ACT = LCPDAT2924
FDAT_ACT = FP2924
BAS(#CP_PARAMS, 2.0)
SET_CD_PARAMS (0)
LIN XP2924
;ENDFOLD

;FOLD LIN P2925 Vel=2 m/s CPDAT2925 Tool[1]:marker Base[0] ;%{PE}
;FOLD Parameters ;%{h}
;Params IlfProvider=kukaroboter.basistech.inlineforms.movement.old; Kuka.IsGlobalPoint=False; Kuka.PointName=P2925; Kuka.BlendingEnabled=False; Kuka.MoveDataName=CPDAT1; Kuka.VelocityPath=2; Kuka.CurrentCDSetIndex=0; Kuka.MovementParameterFieldEnabled=True; IlfCommand=LIN
;ENDFOLD
$BWDSTART = FALSE
LDAT_ACT = LCPDAT2925
FDAT_ACT = FP2925
BAS(#CP_PARAMS, 2.0)
SET_CD_PARAMS (0)
LIN XP2925
;ENDFOLD

;FOLD LIN P2926 Vel=2 m/s CPDAT2926 Tool[1]:marker Base[0] ;%{PE}
;FOLD Parameters ;%{h}
;Params IlfProvider=kukaroboter.basistech.inlineforms.movement.old; Kuka.IsGlobalPoint=False; Kuka.PointName=P2926; Kuka.BlendingEnabled=False; Kuka.MoveDataName=CPDAT1; Kuka.VelocityPath=2; Kuka.CurrentCDSetIndex=0; Kuka.MovementParameterFieldEnabled=True; IlfCommand=LIN
;ENDFOLD
$BWDSTART = FALSE
LDAT_ACT = LCPDAT2926
FDAT_ACT = FP2926
BAS(#CP_PARAMS, 2.0)
SET_CD_PARAMS (0)
LIN XP2926
;ENDFOLD

;FOLD LIN P2927 Vel=2 m/s CPDAT2927 Tool[1]:marker Base[0] ;%{PE}
;FOLD Parameters ;%{h}
;Params IlfProvider=kukaroboter.basistech.inlineforms.movement.old; Kuka.IsGlobalPoint=False; Kuka.PointName=P2927; Kuka.BlendingEnabled=False; Kuka.MoveDataName=CPDAT1; Kuka.VelocityPath=2; Kuka.CurrentCDSetIndex=0; Kuka.MovementParameterFieldEnabled=True; IlfCommand=LIN
;ENDFOLD
$BWDSTART = FALSE
LDAT_ACT = LCPDAT2927
FDAT_ACT = FP2927
BAS(#CP_PARAMS, 2.0)
SET_CD_PARAMS (0)
LIN XP2927
;ENDFOLD

;FOLD LIN P2928 Vel=2 m/s CPDAT2928 Tool[1]:marker Base[0] ;%{PE}
;FOLD Parameters ;%{h}
;Params IlfProvider=kukaroboter.basistech.inlineforms.movement.old; Kuka.IsGlobalPoint=False; Kuka.PointName=P2928; Kuka.BlendingEnabled=False; Kuka.MoveDataName=CPDAT1; Kuka.VelocityPath=2; Kuka.CurrentCDSetIndex=0; Kuka.MovementParameterFieldEnabled=True; IlfCommand=LIN
;ENDFOLD
$BWDSTART = FALSE
LDAT_ACT = LCPDAT2928
FDAT_ACT = FP2928
BAS(#CP_PARAMS, 2.0)
SET_CD_PARAMS (0)
LIN XP2928
;ENDFOLD

;FOLD LIN P2929 Vel=2 m/s CPDAT2929 Tool[1]:marker Base[0] ;%{PE}
;FOLD Parameters ;%{h}
;Params IlfProvider=kukaroboter.basistech.inlineforms.movement.old; Kuka.IsGlobalPoint=False; Kuka.PointName=P2929; Kuka.BlendingEnabled=False; Kuka.MoveDataName=CPDAT1; Kuka.VelocityPath=2; Kuka.CurrentCDSetIndex=0; Kuka.MovementParameterFieldEnabled=True; IlfCommand=LIN
;ENDFOLD
$BWDSTART = FALSE
LDAT_ACT = LCPDAT2929
FDAT_ACT = FP2929
BAS(#CP_PARAMS, 2.0)
SET_CD_PARAMS (0)
LIN XP2929
;ENDFOLD

;FOLD LIN P2930 Vel=2 m/s CPDAT2930 Tool[1]:marker Base[0] ;%{PE}
;FOLD Parameters ;%{h}
;Params IlfProvider=kukaroboter.basistech.inlineforms.movement.old; Kuka.IsGlobalPoint=False; Kuka.PointName=P2930; Kuka.BlendingEnabled=False; Kuka.MoveDataName=CPDAT1; Kuka.VelocityPath=2; Kuka.CurrentCDSetIndex=0; Kuka.MovementParameterFieldEnabled=True; IlfCommand=LIN
;ENDFOLD
$BWDSTART = FALSE
LDAT_ACT = LCPDAT2930
FDAT_ACT = FP2930
BAS(#CP_PARAMS, 2.0)
SET_CD_PARAMS (0)
LIN XP2930
;ENDFOLD

;FOLD LIN P2931 Vel=2 m/s CPDAT2931 Tool[1]:marker Base[0] ;%{PE}
;FOLD Parameters ;%{h}
;Params IlfProvider=kukaroboter.basistech.inlineforms.movement.old; Kuka.IsGlobalPoint=False; Kuka.PointName=P2931; Kuka.BlendingEnabled=False; Kuka.MoveDataName=CPDAT1; Kuka.VelocityPath=2; Kuka.CurrentCDSetIndex=0; Kuka.MovementParameterFieldEnabled=True; IlfCommand=LIN
;ENDFOLD
$BWDSTART = FALSE
LDAT_ACT = LCPDAT2931
FDAT_ACT = FP2931
BAS(#CP_PARAMS, 2.0)
SET_CD_PARAMS (0)
LIN XP2931
;ENDFOLD

;FOLD LIN P2932 Vel=2 m/s CPDAT2932 Tool[1]:marker Base[0] ;%{PE}
;FOLD Parameters ;%{h}
;Params IlfProvider=kukaroboter.basistech.inlineforms.movement.old; Kuka.IsGlobalPoint=False; Kuka.PointName=P2932; Kuka.BlendingEnabled=False; Kuka.MoveDataName=CPDAT1; Kuka.VelocityPath=2; Kuka.CurrentCDSetIndex=0; Kuka.MovementParameterFieldEnabled=True; IlfCommand=LIN
;ENDFOLD
$BWDSTART = FALSE
LDAT_ACT = LCPDAT2932
FDAT_ACT = FP2932
BAS(#CP_PARAMS, 2.0)
SET_CD_PARAMS (0)
LIN XP2932
;ENDFOLD

;FOLD LIN P2933 Vel=2 m/s CPDAT2933 Tool[1]:marker Base[0] ;%{PE}
;FOLD Parameters ;%{h}
;Params IlfProvider=kukaroboter.basistech.inlineforms.movement.old; Kuka.IsGlobalPoint=False; Kuka.PointName=P2933; Kuka.BlendingEnabled=False; Kuka.MoveDataName=CPDAT1; Kuka.VelocityPath=2; Kuka.CurrentCDSetIndex=0; Kuka.MovementParameterFieldEnabled=True; IlfCommand=LIN
;ENDFOLD
$BWDSTART = FALSE
LDAT_ACT = LCPDAT2933
FDAT_ACT = FP2933
BAS(#CP_PARAMS, 2.0)
SET_CD_PARAMS (0)
LIN XP2933
;ENDFOLD

;FOLD LIN P2934 Vel=2 m/s CPDAT2934 Tool[1]:marker Base[0] ;%{PE}
;FOLD Parameters ;%{h}
;Params IlfProvider=kukaroboter.basistech.inlineforms.movement.old; Kuka.IsGlobalPoint=False; Kuka.PointName=P2934; Kuka.BlendingEnabled=False; Kuka.MoveDataName=CPDAT1; Kuka.VelocityPath=2; Kuka.CurrentCDSetIndex=0; Kuka.MovementParameterFieldEnabled=True; IlfCommand=LIN
;ENDFOLD
$BWDSTART = FALSE
LDAT_ACT = LCPDAT2934
FDAT_ACT = FP2934
BAS(#CP_PARAMS, 2.0)
SET_CD_PARAMS (0)
LIN XP2934
;ENDFOLD

;FOLD LIN P2935 Vel=2 m/s CPDAT2935 Tool[1]:marker Base[0] ;%{PE}
;FOLD Parameters ;%{h}
;Params IlfProvider=kukaroboter.basistech.inlineforms.movement.old; Kuka.IsGlobalPoint=False; Kuka.PointName=P2935; Kuka.BlendingEnabled=False; Kuka.MoveDataName=CPDAT1; Kuka.VelocityPath=2; Kuka.CurrentCDSetIndex=0; Kuka.MovementParameterFieldEnabled=True; IlfCommand=LIN
;ENDFOLD
$BWDSTART = FALSE
LDAT_ACT = LCPDAT2935
FDAT_ACT = FP2935
BAS(#CP_PARAMS, 2.0)
SET_CD_PARAMS (0)
LIN XP2935
;ENDFOLD

;FOLD LIN P2936 Vel=2 m/s CPDAT2936 Tool[1]:marker Base[0] ;%{PE}
;FOLD Parameters ;%{h}
;Params IlfProvider=kukaroboter.basistech.inlineforms.movement.old; Kuka.IsGlobalPoint=False; Kuka.PointName=P2936; Kuka.BlendingEnabled=False; Kuka.MoveDataName=CPDAT1; Kuka.VelocityPath=2; Kuka.CurrentCDSetIndex=0; Kuka.MovementParameterFieldEnabled=True; IlfCommand=LIN
;ENDFOLD
$BWDSTART = FALSE
LDAT_ACT = LCPDAT2936
FDAT_ACT = FP2936
BAS(#CP_PARAMS, 2.0)
SET_CD_PARAMS (0)
LIN XP2936
;ENDFOLD

;FOLD LIN P2937 Vel=2 m/s CPDAT2937 Tool[1]:marker Base[0] ;%{PE}
;FOLD Parameters ;%{h}
;Params IlfProvider=kukaroboter.basistech.inlineforms.movement.old; Kuka.IsGlobalPoint=False; Kuka.PointName=P2937; Kuka.BlendingEnabled=False; Kuka.MoveDataName=CPDAT1; Kuka.VelocityPath=2; Kuka.CurrentCDSetIndex=0; Kuka.MovementParameterFieldEnabled=True; IlfCommand=LIN
;ENDFOLD
$BWDSTART = FALSE
LDAT_ACT = LCPDAT2937
FDAT_ACT = FP2937
BAS(#CP_PARAMS, 2.0)
SET_CD_PARAMS (0)
LIN XP2937
;ENDFOLD

;FOLD LIN P2938 Vel=2 m/s CPDAT2938 Tool[1]:marker Base[0] ;%{PE}
;FOLD Parameters ;%{h}
;Params IlfProvider=kukaroboter.basistech.inlineforms.movement.old; Kuka.IsGlobalPoint=False; Kuka.PointName=P2938; Kuka.BlendingEnabled=False; Kuka.MoveDataName=CPDAT1; Kuka.VelocityPath=2; Kuka.CurrentCDSetIndex=0; Kuka.MovementParameterFieldEnabled=True; IlfCommand=LIN
;ENDFOLD
$BWDSTART = FALSE
LDAT_ACT = LCPDAT2938
FDAT_ACT = FP2938
BAS(#CP_PARAMS, 2.0)
SET_CD_PARAMS (0)
LIN XP2938
;ENDFOLD

;FOLD LIN P2939 Vel=2 m/s CPDAT2939 Tool[1]:marker Base[0] ;%{PE}
;FOLD Parameters ;%{h}
;Params IlfProvider=kukaroboter.basistech.inlineforms.movement.old; Kuka.IsGlobalPoint=False; Kuka.PointName=P2939; Kuka.BlendingEnabled=False; Kuka.MoveDataName=CPDAT1; Kuka.VelocityPath=2; Kuka.CurrentCDSetIndex=0; Kuka.MovementParameterFieldEnabled=True; IlfCommand=LIN
;ENDFOLD
$BWDSTART = FALSE
LDAT_ACT = LCPDAT2939
FDAT_ACT = FP2939
BAS(#CP_PARAMS, 2.0)
SET_CD_PARAMS (0)
LIN XP2939
;ENDFOLD

;FOLD LIN P2940 Vel=2 m/s CPDAT2940 Tool[1]:marker Base[0] ;%{PE}
;FOLD Parameters ;%{h}
;Params IlfProvider=kukaroboter.basistech.inlineforms.movement.old; Kuka.IsGlobalPoint=False; Kuka.PointName=P2940; Kuka.BlendingEnabled=False; Kuka.MoveDataName=CPDAT1; Kuka.VelocityPath=2; Kuka.CurrentCDSetIndex=0; Kuka.MovementParameterFieldEnabled=True; IlfCommand=LIN
;ENDFOLD
$BWDSTART = FALSE
LDAT_ACT = LCPDAT2940
FDAT_ACT = FP2940
BAS(#CP_PARAMS, 2.0)
SET_CD_PARAMS (0)
LIN XP2940
;ENDFOLD

;FOLD LIN P2941 Vel=2 m/s CPDAT2941 Tool[1]:marker Base[0] ;%{PE}
;FOLD Parameters ;%{h}
;Params IlfProvider=kukaroboter.basistech.inlineforms.movement.old; Kuka.IsGlobalPoint=False; Kuka.PointName=P2941; Kuka.BlendingEnabled=False; Kuka.MoveDataName=CPDAT1; Kuka.VelocityPath=2; Kuka.CurrentCDSetIndex=0; Kuka.MovementParameterFieldEnabled=True; IlfCommand=LIN
;ENDFOLD
$BWDSTART = FALSE
LDAT_ACT = LCPDAT2941
FDAT_ACT = FP2941
BAS(#CP_PARAMS, 2.0)
SET_CD_PARAMS (0)
LIN XP2941
;ENDFOLD

;FOLD LIN P2942 Vel=2 m/s CPDAT2942 Tool[1]:marker Base[0] ;%{PE}
;FOLD Parameters ;%{h}
;Params IlfProvider=kukaroboter.basistech.inlineforms.movement.old; Kuka.IsGlobalPoint=False; Kuka.PointName=P2942; Kuka.BlendingEnabled=False; Kuka.MoveDataName=CPDAT1; Kuka.VelocityPath=2; Kuka.CurrentCDSetIndex=0; Kuka.MovementParameterFieldEnabled=True; IlfCommand=LIN
;ENDFOLD
$BWDSTART = FALSE
LDAT_ACT = LCPDAT2942
FDAT_ACT = FP2942
BAS(#CP_PARAMS, 2.0)
SET_CD_PARAMS (0)
LIN XP2942
;ENDFOLD

;FOLD LIN P2943 Vel=2 m/s CPDAT2943 Tool[1]:marker Base[0] ;%{PE}
;FOLD Parameters ;%{h}
;Params IlfProvider=kukaroboter.basistech.inlineforms.movement.old; Kuka.IsGlobalPoint=False; Kuka.PointName=P2943; Kuka.BlendingEnabled=False; Kuka.MoveDataName=CPDAT1; Kuka.VelocityPath=2; Kuka.CurrentCDSetIndex=0; Kuka.MovementParameterFieldEnabled=True; IlfCommand=LIN
;ENDFOLD
$BWDSTART = FALSE
LDAT_ACT = LCPDAT2943
FDAT_ACT = FP2943
BAS(#CP_PARAMS, 2.0)
SET_CD_PARAMS (0)
LIN XP2943
;ENDFOLD

;FOLD LIN P2944 Vel=2 m/s CPDAT2944 Tool[1]:marker Base[0] ;%{PE}
;FOLD Parameters ;%{h}
;Params IlfProvider=kukaroboter.basistech.inlineforms.movement.old; Kuka.IsGlobalPoint=False; Kuka.PointName=P2944; Kuka.BlendingEnabled=False; Kuka.MoveDataName=CPDAT1; Kuka.VelocityPath=2; Kuka.CurrentCDSetIndex=0; Kuka.MovementParameterFieldEnabled=True; IlfCommand=LIN
;ENDFOLD
$BWDSTART = FALSE
LDAT_ACT = LCPDAT2944
FDAT_ACT = FP2944
BAS(#CP_PARAMS, 2.0)
SET_CD_PARAMS (0)
LIN XP2944
;ENDFOLD

;FOLD LIN P2945 Vel=2 m/s CPDAT2945 Tool[1]:marker Base[0] ;%{PE}
;FOLD Parameters ;%{h}
;Params IlfProvider=kukaroboter.basistech.inlineforms.movement.old; Kuka.IsGlobalPoint=False; Kuka.PointName=P2945; Kuka.BlendingEnabled=False; Kuka.MoveDataName=CPDAT1; Kuka.VelocityPath=2; Kuka.CurrentCDSetIndex=0; Kuka.MovementParameterFieldEnabled=True; IlfCommand=LIN
;ENDFOLD
$BWDSTART = FALSE
LDAT_ACT = LCPDAT2945
FDAT_ACT = FP2945
BAS(#CP_PARAMS, 2.0)
SET_CD_PARAMS (0)
LIN XP2945
;ENDFOLD

;FOLD LIN P2946 Vel=2 m/s CPDAT2946 Tool[1]:marker Base[0] ;%{PE}
;FOLD Parameters ;%{h}
;Params IlfProvider=kukaroboter.basistech.inlineforms.movement.old; Kuka.IsGlobalPoint=False; Kuka.PointName=P2946; Kuka.BlendingEnabled=False; Kuka.MoveDataName=CPDAT1; Kuka.VelocityPath=2; Kuka.CurrentCDSetIndex=0; Kuka.MovementParameterFieldEnabled=True; IlfCommand=LIN
;ENDFOLD
$BWDSTART = FALSE
LDAT_ACT = LCPDAT2946
FDAT_ACT = FP2946
BAS(#CP_PARAMS, 2.0)
SET_CD_PARAMS (0)
LIN XP2946
;ENDFOLD

;FOLD LIN P2947 Vel=2 m/s CPDAT2947 Tool[1]:marker Base[0] ;%{PE}
;FOLD Parameters ;%{h}
;Params IlfProvider=kukaroboter.basistech.inlineforms.movement.old; Kuka.IsGlobalPoint=False; Kuka.PointName=P2947; Kuka.BlendingEnabled=False; Kuka.MoveDataName=CPDAT1; Kuka.VelocityPath=2; Kuka.CurrentCDSetIndex=0; Kuka.MovementParameterFieldEnabled=True; IlfCommand=LIN
;ENDFOLD
$BWDSTART = FALSE
LDAT_ACT = LCPDAT2947
FDAT_ACT = FP2947
BAS(#CP_PARAMS, 2.0)
SET_CD_PARAMS (0)
LIN XP2947
;ENDFOLD

;FOLD LIN P2948 Vel=2 m/s CPDAT2948 Tool[1]:marker Base[0] ;%{PE}
;FOLD Parameters ;%{h}
;Params IlfProvider=kukaroboter.basistech.inlineforms.movement.old; Kuka.IsGlobalPoint=False; Kuka.PointName=P2948; Kuka.BlendingEnabled=False; Kuka.MoveDataName=CPDAT1; Kuka.VelocityPath=2; Kuka.CurrentCDSetIndex=0; Kuka.MovementParameterFieldEnabled=True; IlfCommand=LIN
;ENDFOLD
$BWDSTART = FALSE
LDAT_ACT = LCPDAT2948
FDAT_ACT = FP2948
BAS(#CP_PARAMS, 2.0)
SET_CD_PARAMS (0)
LIN XP2948
;ENDFOLD

;FOLD LIN P2949 Vel=2 m/s CPDAT2949 Tool[1]:marker Base[0] ;%{PE}
;FOLD Parameters ;%{h}
;Params IlfProvider=kukaroboter.basistech.inlineforms.movement.old; Kuka.IsGlobalPoint=False; Kuka.PointName=P2949; Kuka.BlendingEnabled=False; Kuka.MoveDataName=CPDAT1; Kuka.VelocityPath=2; Kuka.CurrentCDSetIndex=0; Kuka.MovementParameterFieldEnabled=True; IlfCommand=LIN
;ENDFOLD
$BWDSTART = FALSE
LDAT_ACT = LCPDAT2949
FDAT_ACT = FP2949
BAS(#CP_PARAMS, 2.0)
SET_CD_PARAMS (0)
LIN XP2949
;ENDFOLD

;FOLD LIN P2950 Vel=2 m/s CPDAT2950 Tool[1]:marker Base[0] ;%{PE}
;FOLD Parameters ;%{h}
;Params IlfProvider=kukaroboter.basistech.inlineforms.movement.old; Kuka.IsGlobalPoint=False; Kuka.PointName=P2950; Kuka.BlendingEnabled=False; Kuka.MoveDataName=CPDAT1; Kuka.VelocityPath=2; Kuka.CurrentCDSetIndex=0; Kuka.MovementParameterFieldEnabled=True; IlfCommand=LIN
;ENDFOLD
$BWDSTART = FALSE
LDAT_ACT = LCPDAT2950
FDAT_ACT = FP2950
BAS(#CP_PARAMS, 2.0)
SET_CD_PARAMS (0)
LIN XP2950
;ENDFOLD

;FOLD LIN P2951 Vel=2 m/s CPDAT2951 Tool[1]:marker Base[0] ;%{PE}
;FOLD Parameters ;%{h}
;Params IlfProvider=kukaroboter.basistech.inlineforms.movement.old; Kuka.IsGlobalPoint=False; Kuka.PointName=P2951; Kuka.BlendingEnabled=False; Kuka.MoveDataName=CPDAT1; Kuka.VelocityPath=2; Kuka.CurrentCDSetIndex=0; Kuka.MovementParameterFieldEnabled=True; IlfCommand=LIN
;ENDFOLD
$BWDSTART = FALSE
LDAT_ACT = LCPDAT2951
FDAT_ACT = FP2951
BAS(#CP_PARAMS, 2.0)
SET_CD_PARAMS (0)
LIN XP2951
;ENDFOLD

;FOLD LIN P2952 Vel=2 m/s CPDAT2952 Tool[1]:marker Base[0] ;%{PE}
;FOLD Parameters ;%{h}
;Params IlfProvider=kukaroboter.basistech.inlineforms.movement.old; Kuka.IsGlobalPoint=False; Kuka.PointName=P2952; Kuka.BlendingEnabled=False; Kuka.MoveDataName=CPDAT1; Kuka.VelocityPath=2; Kuka.CurrentCDSetIndex=0; Kuka.MovementParameterFieldEnabled=True; IlfCommand=LIN
;ENDFOLD
$BWDSTART = FALSE
LDAT_ACT = LCPDAT2952
FDAT_ACT = FP2952
BAS(#CP_PARAMS, 2.0)
SET_CD_PARAMS (0)
LIN XP2952
;ENDFOLD

;FOLD LIN P2953 Vel=2 m/s CPDAT2953 Tool[1]:marker Base[0] ;%{PE}
;FOLD Parameters ;%{h}
;Params IlfProvider=kukaroboter.basistech.inlineforms.movement.old; Kuka.IsGlobalPoint=False; Kuka.PointName=P2953; Kuka.BlendingEnabled=False; Kuka.MoveDataName=CPDAT1; Kuka.VelocityPath=2; Kuka.CurrentCDSetIndex=0; Kuka.MovementParameterFieldEnabled=True; IlfCommand=LIN
;ENDFOLD
$BWDSTART = FALSE
LDAT_ACT = LCPDAT2953
FDAT_ACT = FP2953
BAS(#CP_PARAMS, 2.0)
SET_CD_PARAMS (0)
LIN XP2953
;ENDFOLD

;FOLD LIN P2954 Vel=2 m/s CPDAT2954 Tool[1]:marker Base[0] ;%{PE}
;FOLD Parameters ;%{h}
;Params IlfProvider=kukaroboter.basistech.inlineforms.movement.old; Kuka.IsGlobalPoint=False; Kuka.PointName=P2954; Kuka.BlendingEnabled=False; Kuka.MoveDataName=CPDAT1; Kuka.VelocityPath=2; Kuka.CurrentCDSetIndex=0; Kuka.MovementParameterFieldEnabled=True; IlfCommand=LIN
;ENDFOLD
$BWDSTART = FALSE
LDAT_ACT = LCPDAT2954
FDAT_ACT = FP2954
BAS(#CP_PARAMS, 2.0)
SET_CD_PARAMS (0)
LIN XP2954
;ENDFOLD

;FOLD LIN P2955 Vel=2 m/s CPDAT2955 Tool[1]:marker Base[0] ;%{PE}
;FOLD Parameters ;%{h}
;Params IlfProvider=kukaroboter.basistech.inlineforms.movement.old; Kuka.IsGlobalPoint=False; Kuka.PointName=P2955; Kuka.BlendingEnabled=False; Kuka.MoveDataName=CPDAT1; Kuka.VelocityPath=2; Kuka.CurrentCDSetIndex=0; Kuka.MovementParameterFieldEnabled=True; IlfCommand=LIN
;ENDFOLD
$BWDSTART = FALSE
LDAT_ACT = LCPDAT2955
FDAT_ACT = FP2955
BAS(#CP_PARAMS, 2.0)
SET_CD_PARAMS (0)
LIN XP2955
;ENDFOLD

;FOLD LIN P2956 Vel=2 m/s CPDAT2956 Tool[1]:marker Base[0] ;%{PE}
;FOLD Parameters ;%{h}
;Params IlfProvider=kukaroboter.basistech.inlineforms.movement.old; Kuka.IsGlobalPoint=False; Kuka.PointName=P2956; Kuka.BlendingEnabled=False; Kuka.MoveDataName=CPDAT1; Kuka.VelocityPath=2; Kuka.CurrentCDSetIndex=0; Kuka.MovementParameterFieldEnabled=True; IlfCommand=LIN
;ENDFOLD
$BWDSTART = FALSE
LDAT_ACT = LCPDAT2956
FDAT_ACT = FP2956
BAS(#CP_PARAMS, 2.0)
SET_CD_PARAMS (0)
LIN XP2956
;ENDFOLD

;FOLD LIN P2957 Vel=2 m/s CPDAT2957 Tool[1]:marker Base[0] ;%{PE}
;FOLD Parameters ;%{h}
;Params IlfProvider=kukaroboter.basistech.inlineforms.movement.old; Kuka.IsGlobalPoint=False; Kuka.PointName=P2957; Kuka.BlendingEnabled=False; Kuka.MoveDataName=CPDAT1; Kuka.VelocityPath=2; Kuka.CurrentCDSetIndex=0; Kuka.MovementParameterFieldEnabled=True; IlfCommand=LIN
;ENDFOLD
$BWDSTART = FALSE
LDAT_ACT = LCPDAT2957
FDAT_ACT = FP2957
BAS(#CP_PARAMS, 2.0)
SET_CD_PARAMS (0)
LIN XP2957
;ENDFOLD

;FOLD LIN P2958 Vel=2 m/s CPDAT2958 Tool[1]:marker Base[0] ;%{PE}
;FOLD Parameters ;%{h}
;Params IlfProvider=kukaroboter.basistech.inlineforms.movement.old; Kuka.IsGlobalPoint=False; Kuka.PointName=P2958; Kuka.BlendingEnabled=False; Kuka.MoveDataName=CPDAT1; Kuka.VelocityPath=2; Kuka.CurrentCDSetIndex=0; Kuka.MovementParameterFieldEnabled=True; IlfCommand=LIN
;ENDFOLD
$BWDSTART = FALSE
LDAT_ACT = LCPDAT2958
FDAT_ACT = FP2958
BAS(#CP_PARAMS, 2.0)
SET_CD_PARAMS (0)
LIN XP2958
;ENDFOLD

;FOLD LIN P2959 Vel=2 m/s CPDAT2959 Tool[1]:marker Base[0] ;%{PE}
;FOLD Parameters ;%{h}
;Params IlfProvider=kukaroboter.basistech.inlineforms.movement.old; Kuka.IsGlobalPoint=False; Kuka.PointName=P2959; Kuka.BlendingEnabled=False; Kuka.MoveDataName=CPDAT1; Kuka.VelocityPath=2; Kuka.CurrentCDSetIndex=0; Kuka.MovementParameterFieldEnabled=True; IlfCommand=LIN
;ENDFOLD
$BWDSTART = FALSE
LDAT_ACT = LCPDAT2959
FDAT_ACT = FP2959
BAS(#CP_PARAMS, 2.0)
SET_CD_PARAMS (0)
LIN XP2959
;ENDFOLD

;FOLD LIN P2960 Vel=2 m/s CPDAT2960 Tool[1]:marker Base[0] ;%{PE}
;FOLD Parameters ;%{h}
;Params IlfProvider=kukaroboter.basistech.inlineforms.movement.old; Kuka.IsGlobalPoint=False; Kuka.PointName=P2960; Kuka.BlendingEnabled=False; Kuka.MoveDataName=CPDAT1; Kuka.VelocityPath=2; Kuka.CurrentCDSetIndex=0; Kuka.MovementParameterFieldEnabled=True; IlfCommand=LIN
;ENDFOLD
$BWDSTART = FALSE
LDAT_ACT = LCPDAT2960
FDAT_ACT = FP2960
BAS(#CP_PARAMS, 2.0)
SET_CD_PARAMS (0)
LIN XP2960
;ENDFOLD

;FOLD LIN P2961 Vel=2 m/s CPDAT2961 Tool[1]:marker Base[0] ;%{PE}
;FOLD Parameters ;%{h}
;Params IlfProvider=kukaroboter.basistech.inlineforms.movement.old; Kuka.IsGlobalPoint=False; Kuka.PointName=P2961; Kuka.BlendingEnabled=False; Kuka.MoveDataName=CPDAT1; Kuka.VelocityPath=2; Kuka.CurrentCDSetIndex=0; Kuka.MovementParameterFieldEnabled=True; IlfCommand=LIN
;ENDFOLD
$BWDSTART = FALSE
LDAT_ACT = LCPDAT2961
FDAT_ACT = FP2961
BAS(#CP_PARAMS, 2.0)
SET_CD_PARAMS (0)
LIN XP2961
;ENDFOLD

;FOLD LIN P2962 Vel=2 m/s CPDAT2962 Tool[1]:marker Base[0] ;%{PE}
;FOLD Parameters ;%{h}
;Params IlfProvider=kukaroboter.basistech.inlineforms.movement.old; Kuka.IsGlobalPoint=False; Kuka.PointName=P2962; Kuka.BlendingEnabled=False; Kuka.MoveDataName=CPDAT1; Kuka.VelocityPath=2; Kuka.CurrentCDSetIndex=0; Kuka.MovementParameterFieldEnabled=True; IlfCommand=LIN
;ENDFOLD
$BWDSTART = FALSE
LDAT_ACT = LCPDAT2962
FDAT_ACT = FP2962
BAS(#CP_PARAMS, 2.0)
SET_CD_PARAMS (0)
LIN XP2962
;ENDFOLD

;FOLD LIN P2963 Vel=2 m/s CPDAT2963 Tool[1]:marker Base[0] ;%{PE}
;FOLD Parameters ;%{h}
;Params IlfProvider=kukaroboter.basistech.inlineforms.movement.old; Kuka.IsGlobalPoint=False; Kuka.PointName=P2963; Kuka.BlendingEnabled=False; Kuka.MoveDataName=CPDAT1; Kuka.VelocityPath=2; Kuka.CurrentCDSetIndex=0; Kuka.MovementParameterFieldEnabled=True; IlfCommand=LIN
;ENDFOLD
$BWDSTART = FALSE
LDAT_ACT = LCPDAT2963
FDAT_ACT = FP2963
BAS(#CP_PARAMS, 2.0)
SET_CD_PARAMS (0)
LIN XP2963
;ENDFOLD

;FOLD LIN P2964 Vel=2 m/s CPDAT2964 Tool[1]:marker Base[0] ;%{PE}
;FOLD Parameters ;%{h}
;Params IlfProvider=kukaroboter.basistech.inlineforms.movement.old; Kuka.IsGlobalPoint=False; Kuka.PointName=P2964; Kuka.BlendingEnabled=False; Kuka.MoveDataName=CPDAT1; Kuka.VelocityPath=2; Kuka.CurrentCDSetIndex=0; Kuka.MovementParameterFieldEnabled=True; IlfCommand=LIN
;ENDFOLD
$BWDSTART = FALSE
LDAT_ACT = LCPDAT2964
FDAT_ACT = FP2964
BAS(#CP_PARAMS, 2.0)
SET_CD_PARAMS (0)
LIN XP2964
;ENDFOLD

;FOLD LIN P2965 Vel=2 m/s CPDAT2965 Tool[1]:marker Base[0] ;%{PE}
;FOLD Parameters ;%{h}
;Params IlfProvider=kukaroboter.basistech.inlineforms.movement.old; Kuka.IsGlobalPoint=False; Kuka.PointName=P2965; Kuka.BlendingEnabled=False; Kuka.MoveDataName=CPDAT1; Kuka.VelocityPath=2; Kuka.CurrentCDSetIndex=0; Kuka.MovementParameterFieldEnabled=True; IlfCommand=LIN
;ENDFOLD
$BWDSTART = FALSE
LDAT_ACT = LCPDAT2965
FDAT_ACT = FP2965
BAS(#CP_PARAMS, 2.0)
SET_CD_PARAMS (0)
LIN XP2965
;ENDFOLD

;FOLD LIN P2966 Vel=2 m/s CPDAT2966 Tool[1]:marker Base[0] ;%{PE}
;FOLD Parameters ;%{h}
;Params IlfProvider=kukaroboter.basistech.inlineforms.movement.old; Kuka.IsGlobalPoint=False; Kuka.PointName=P2966; Kuka.BlendingEnabled=False; Kuka.MoveDataName=CPDAT1; Kuka.VelocityPath=2; Kuka.CurrentCDSetIndex=0; Kuka.MovementParameterFieldEnabled=True; IlfCommand=LIN
;ENDFOLD
$BWDSTART = FALSE
LDAT_ACT = LCPDAT2966
FDAT_ACT = FP2966
BAS(#CP_PARAMS, 2.0)
SET_CD_PARAMS (0)
LIN XP2966
;ENDFOLD

;FOLD LIN P2967 Vel=2 m/s CPDAT2967 Tool[1]:marker Base[0] ;%{PE}
;FOLD Parameters ;%{h}
;Params IlfProvider=kukaroboter.basistech.inlineforms.movement.old; Kuka.IsGlobalPoint=False; Kuka.PointName=P2967; Kuka.BlendingEnabled=False; Kuka.MoveDataName=CPDAT1; Kuka.VelocityPath=2; Kuka.CurrentCDSetIndex=0; Kuka.MovementParameterFieldEnabled=True; IlfCommand=LIN
;ENDFOLD
$BWDSTART = FALSE
LDAT_ACT = LCPDAT2967
FDAT_ACT = FP2967
BAS(#CP_PARAMS, 2.0)
SET_CD_PARAMS (0)
LIN XP2967
;ENDFOLD

;FOLD LIN P2968 Vel=2 m/s CPDAT2968 Tool[1]:marker Base[0] ;%{PE}
;FOLD Parameters ;%{h}
;Params IlfProvider=kukaroboter.basistech.inlineforms.movement.old; Kuka.IsGlobalPoint=False; Kuka.PointName=P2968; Kuka.BlendingEnabled=False; Kuka.MoveDataName=CPDAT1; Kuka.VelocityPath=2; Kuka.CurrentCDSetIndex=0; Kuka.MovementParameterFieldEnabled=True; IlfCommand=LIN
;ENDFOLD
$BWDSTART = FALSE
LDAT_ACT = LCPDAT2968
FDAT_ACT = FP2968
BAS(#CP_PARAMS, 2.0)
SET_CD_PARAMS (0)
LIN XP2968
;ENDFOLD

;FOLD LIN P2969 Vel=2 m/s CPDAT2969 Tool[1]:marker Base[0] ;%{PE}
;FOLD Parameters ;%{h}
;Params IlfProvider=kukaroboter.basistech.inlineforms.movement.old; Kuka.IsGlobalPoint=False; Kuka.PointName=P2969; Kuka.BlendingEnabled=False; Kuka.MoveDataName=CPDAT1; Kuka.VelocityPath=2; Kuka.CurrentCDSetIndex=0; Kuka.MovementParameterFieldEnabled=True; IlfCommand=LIN
;ENDFOLD
$BWDSTART = FALSE
LDAT_ACT = LCPDAT2969
FDAT_ACT = FP2969
BAS(#CP_PARAMS, 2.0)
SET_CD_PARAMS (0)
LIN XP2969
;ENDFOLD

;FOLD LIN P2970 Vel=2 m/s CPDAT2970 Tool[1]:marker Base[0] ;%{PE}
;FOLD Parameters ;%{h}
;Params IlfProvider=kukaroboter.basistech.inlineforms.movement.old; Kuka.IsGlobalPoint=False; Kuka.PointName=P2970; Kuka.BlendingEnabled=False; Kuka.MoveDataName=CPDAT1; Kuka.VelocityPath=2; Kuka.CurrentCDSetIndex=0; Kuka.MovementParameterFieldEnabled=True; IlfCommand=LIN
;ENDFOLD
$BWDSTART = FALSE
LDAT_ACT = LCPDAT2970
FDAT_ACT = FP2970
BAS(#CP_PARAMS, 2.0)
SET_CD_PARAMS (0)
LIN XP2970
;ENDFOLD

;FOLD LIN P2971 Vel=2 m/s CPDAT2971 Tool[1]:marker Base[0] ;%{PE}
;FOLD Parameters ;%{h}
;Params IlfProvider=kukaroboter.basistech.inlineforms.movement.old; Kuka.IsGlobalPoint=False; Kuka.PointName=P2971; Kuka.BlendingEnabled=False; Kuka.MoveDataName=CPDAT1; Kuka.VelocityPath=2; Kuka.CurrentCDSetIndex=0; Kuka.MovementParameterFieldEnabled=True; IlfCommand=LIN
;ENDFOLD
$BWDSTART = FALSE
LDAT_ACT = LCPDAT2971
FDAT_ACT = FP2971
BAS(#CP_PARAMS, 2.0)
SET_CD_PARAMS (0)
LIN XP2971
;ENDFOLD

;FOLD LIN P2972 Vel=2 m/s CPDAT2972 Tool[1]:marker Base[0] ;%{PE}
;FOLD Parameters ;%{h}
;Params IlfProvider=kukaroboter.basistech.inlineforms.movement.old; Kuka.IsGlobalPoint=False; Kuka.PointName=P2972; Kuka.BlendingEnabled=False; Kuka.MoveDataName=CPDAT1; Kuka.VelocityPath=2; Kuka.CurrentCDSetIndex=0; Kuka.MovementParameterFieldEnabled=True; IlfCommand=LIN
;ENDFOLD
$BWDSTART = FALSE
LDAT_ACT = LCPDAT2972
FDAT_ACT = FP2972
BAS(#CP_PARAMS, 2.0)
SET_CD_PARAMS (0)
LIN XP2972
;ENDFOLD

;FOLD LIN P2973 Vel=2 m/s CPDAT2973 Tool[1]:marker Base[0] ;%{PE}
;FOLD Parameters ;%{h}
;Params IlfProvider=kukaroboter.basistech.inlineforms.movement.old; Kuka.IsGlobalPoint=False; Kuka.PointName=P2973; Kuka.BlendingEnabled=False; Kuka.MoveDataName=CPDAT1; Kuka.VelocityPath=2; Kuka.CurrentCDSetIndex=0; Kuka.MovementParameterFieldEnabled=True; IlfCommand=LIN
;ENDFOLD
$BWDSTART = FALSE
LDAT_ACT = LCPDAT2973
FDAT_ACT = FP2973
BAS(#CP_PARAMS, 2.0)
SET_CD_PARAMS (0)
LIN XP2973
;ENDFOLD

;FOLD LIN P2974 Vel=2 m/s CPDAT2974 Tool[1]:marker Base[0] ;%{PE}
;FOLD Parameters ;%{h}
;Params IlfProvider=kukaroboter.basistech.inlineforms.movement.old; Kuka.IsGlobalPoint=False; Kuka.PointName=P2974; Kuka.BlendingEnabled=False; Kuka.MoveDataName=CPDAT1; Kuka.VelocityPath=2; Kuka.CurrentCDSetIndex=0; Kuka.MovementParameterFieldEnabled=True; IlfCommand=LIN
;ENDFOLD
$BWDSTART = FALSE
LDAT_ACT = LCPDAT2974
FDAT_ACT = FP2974
BAS(#CP_PARAMS, 2.0)
SET_CD_PARAMS (0)
LIN XP2974
;ENDFOLD

;FOLD LIN P2975 Vel=2 m/s CPDAT2975 Tool[1]:marker Base[0] ;%{PE}
;FOLD Parameters ;%{h}
;Params IlfProvider=kukaroboter.basistech.inlineforms.movement.old; Kuka.IsGlobalPoint=False; Kuka.PointName=P2975; Kuka.BlendingEnabled=False; Kuka.MoveDataName=CPDAT1; Kuka.VelocityPath=2; Kuka.CurrentCDSetIndex=0; Kuka.MovementParameterFieldEnabled=True; IlfCommand=LIN
;ENDFOLD
$BWDSTART = FALSE
LDAT_ACT = LCPDAT2975
FDAT_ACT = FP2975
BAS(#CP_PARAMS, 2.0)
SET_CD_PARAMS (0)
LIN XP2975
;ENDFOLD

;FOLD LIN P2976 Vel=2 m/s CPDAT2976 Tool[1]:marker Base[0] ;%{PE}
;FOLD Parameters ;%{h}
;Params IlfProvider=kukaroboter.basistech.inlineforms.movement.old; Kuka.IsGlobalPoint=False; Kuka.PointName=P2976; Kuka.BlendingEnabled=False; Kuka.MoveDataName=CPDAT1; Kuka.VelocityPath=2; Kuka.CurrentCDSetIndex=0; Kuka.MovementParameterFieldEnabled=True; IlfCommand=LIN
;ENDFOLD
$BWDSTART = FALSE
LDAT_ACT = LCPDAT2976
FDAT_ACT = FP2976
BAS(#CP_PARAMS, 2.0)
SET_CD_PARAMS (0)
LIN XP2976
;ENDFOLD

;FOLD LIN P2977 Vel=2 m/s CPDAT2977 Tool[1]:marker Base[0] ;%{PE}
;FOLD Parameters ;%{h}
;Params IlfProvider=kukaroboter.basistech.inlineforms.movement.old; Kuka.IsGlobalPoint=False; Kuka.PointName=P2977; Kuka.BlendingEnabled=False; Kuka.MoveDataName=CPDAT1; Kuka.VelocityPath=2; Kuka.CurrentCDSetIndex=0; Kuka.MovementParameterFieldEnabled=True; IlfCommand=LIN
;ENDFOLD
$BWDSTART = FALSE
LDAT_ACT = LCPDAT2977
FDAT_ACT = FP2977
BAS(#CP_PARAMS, 2.0)
SET_CD_PARAMS (0)
LIN XP2977
;ENDFOLD

;FOLD LIN P2978 Vel=2 m/s CPDAT2978 Tool[1]:marker Base[0] ;%{PE}
;FOLD Parameters ;%{h}
;Params IlfProvider=kukaroboter.basistech.inlineforms.movement.old; Kuka.IsGlobalPoint=False; Kuka.PointName=P2978; Kuka.BlendingEnabled=False; Kuka.MoveDataName=CPDAT1; Kuka.VelocityPath=2; Kuka.CurrentCDSetIndex=0; Kuka.MovementParameterFieldEnabled=True; IlfCommand=LIN
;ENDFOLD
$BWDSTART = FALSE
LDAT_ACT = LCPDAT2978
FDAT_ACT = FP2978
BAS(#CP_PARAMS, 2.0)
SET_CD_PARAMS (0)
LIN XP2978
;ENDFOLD

;FOLD LIN P2979 Vel=2 m/s CPDAT2979 Tool[1]:marker Base[0] ;%{PE}
;FOLD Parameters ;%{h}
;Params IlfProvider=kukaroboter.basistech.inlineforms.movement.old; Kuka.IsGlobalPoint=False; Kuka.PointName=P2979; Kuka.BlendingEnabled=False; Kuka.MoveDataName=CPDAT1; Kuka.VelocityPath=2; Kuka.CurrentCDSetIndex=0; Kuka.MovementParameterFieldEnabled=True; IlfCommand=LIN
;ENDFOLD
$BWDSTART = FALSE
LDAT_ACT = LCPDAT2979
FDAT_ACT = FP2979
BAS(#CP_PARAMS, 2.0)
SET_CD_PARAMS (0)
LIN XP2979
;ENDFOLD

;FOLD LIN P2980 Vel=2 m/s CPDAT2980 Tool[1]:marker Base[0] ;%{PE}
;FOLD Parameters ;%{h}
;Params IlfProvider=kukaroboter.basistech.inlineforms.movement.old; Kuka.IsGlobalPoint=False; Kuka.PointName=P2980; Kuka.BlendingEnabled=False; Kuka.MoveDataName=CPDAT1; Kuka.VelocityPath=2; Kuka.CurrentCDSetIndex=0; Kuka.MovementParameterFieldEnabled=True; IlfCommand=LIN
;ENDFOLD
$BWDSTART = FALSE
LDAT_ACT = LCPDAT2980
FDAT_ACT = FP2980
BAS(#CP_PARAMS, 2.0)
SET_CD_PARAMS (0)
LIN XP2980
;ENDFOLD

;FOLD LIN P2981 Vel=2 m/s CPDAT2981 Tool[1]:marker Base[0] ;%{PE}
;FOLD Parameters ;%{h}
;Params IlfProvider=kukaroboter.basistech.inlineforms.movement.old; Kuka.IsGlobalPoint=False; Kuka.PointName=P2981; Kuka.BlendingEnabled=False; Kuka.MoveDataName=CPDAT1; Kuka.VelocityPath=2; Kuka.CurrentCDSetIndex=0; Kuka.MovementParameterFieldEnabled=True; IlfCommand=LIN
;ENDFOLD
$BWDSTART = FALSE
LDAT_ACT = LCPDAT2981
FDAT_ACT = FP2981
BAS(#CP_PARAMS, 2.0)
SET_CD_PARAMS (0)
LIN XP2981
;ENDFOLD

;FOLD LIN P2982 Vel=2 m/s CPDAT2982 Tool[1]:marker Base[0] ;%{PE}
;FOLD Parameters ;%{h}
;Params IlfProvider=kukaroboter.basistech.inlineforms.movement.old; Kuka.IsGlobalPoint=False; Kuka.PointName=P2982; Kuka.BlendingEnabled=False; Kuka.MoveDataName=CPDAT1; Kuka.VelocityPath=2; Kuka.CurrentCDSetIndex=0; Kuka.MovementParameterFieldEnabled=True; IlfCommand=LIN
;ENDFOLD
$BWDSTART = FALSE
LDAT_ACT = LCPDAT2982
FDAT_ACT = FP2982
BAS(#CP_PARAMS, 2.0)
SET_CD_PARAMS (0)
LIN XP2982
;ENDFOLD

;FOLD LIN P2983 Vel=2 m/s CPDAT2983 Tool[1]:marker Base[0] ;%{PE}
;FOLD Parameters ;%{h}
;Params IlfProvider=kukaroboter.basistech.inlineforms.movement.old; Kuka.IsGlobalPoint=False; Kuka.PointName=P2983; Kuka.BlendingEnabled=False; Kuka.MoveDataName=CPDAT1; Kuka.VelocityPath=2; Kuka.CurrentCDSetIndex=0; Kuka.MovementParameterFieldEnabled=True; IlfCommand=LIN
;ENDFOLD
$BWDSTART = FALSE
LDAT_ACT = LCPDAT2983
FDAT_ACT = FP2983
BAS(#CP_PARAMS, 2.0)
SET_CD_PARAMS (0)
LIN XP2983
;ENDFOLD

;FOLD LIN P2984 Vel=2 m/s CPDAT2984 Tool[1]:marker Base[0] ;%{PE}
;FOLD Parameters ;%{h}
;Params IlfProvider=kukaroboter.basistech.inlineforms.movement.old; Kuka.IsGlobalPoint=False; Kuka.PointName=P2984; Kuka.BlendingEnabled=False; Kuka.MoveDataName=CPDAT1; Kuka.VelocityPath=2; Kuka.CurrentCDSetIndex=0; Kuka.MovementParameterFieldEnabled=True; IlfCommand=LIN
;ENDFOLD
$BWDSTART = FALSE
LDAT_ACT = LCPDAT2984
FDAT_ACT = FP2984
BAS(#CP_PARAMS, 2.0)
SET_CD_PARAMS (0)
LIN XP2984
;ENDFOLD

;FOLD LIN P2985 Vel=2 m/s CPDAT2985 Tool[1]:marker Base[0] ;%{PE}
;FOLD Parameters ;%{h}
;Params IlfProvider=kukaroboter.basistech.inlineforms.movement.old; Kuka.IsGlobalPoint=False; Kuka.PointName=P2985; Kuka.BlendingEnabled=False; Kuka.MoveDataName=CPDAT1; Kuka.VelocityPath=2; Kuka.CurrentCDSetIndex=0; Kuka.MovementParameterFieldEnabled=True; IlfCommand=LIN
;ENDFOLD
$BWDSTART = FALSE
LDAT_ACT = LCPDAT2985
FDAT_ACT = FP2985
BAS(#CP_PARAMS, 2.0)
SET_CD_PARAMS (0)
LIN XP2985
;ENDFOLD

;FOLD LIN P2986 Vel=2 m/s CPDAT2986 Tool[1]:marker Base[0] ;%{PE}
;FOLD Parameters ;%{h}
;Params IlfProvider=kukaroboter.basistech.inlineforms.movement.old; Kuka.IsGlobalPoint=False; Kuka.PointName=P2986; Kuka.BlendingEnabled=False; Kuka.MoveDataName=CPDAT1; Kuka.VelocityPath=2; Kuka.CurrentCDSetIndex=0; Kuka.MovementParameterFieldEnabled=True; IlfCommand=LIN
;ENDFOLD
$BWDSTART = FALSE
LDAT_ACT = LCPDAT2986
FDAT_ACT = FP2986
BAS(#CP_PARAMS, 2.0)
SET_CD_PARAMS (0)
LIN XP2986
;ENDFOLD

;FOLD LIN P2987 Vel=2 m/s CPDAT2987 Tool[1]:marker Base[0] ;%{PE}
;FOLD Parameters ;%{h}
;Params IlfProvider=kukaroboter.basistech.inlineforms.movement.old; Kuka.IsGlobalPoint=False; Kuka.PointName=P2987; Kuka.BlendingEnabled=False; Kuka.MoveDataName=CPDAT1; Kuka.VelocityPath=2; Kuka.CurrentCDSetIndex=0; Kuka.MovementParameterFieldEnabled=True; IlfCommand=LIN
;ENDFOLD
$BWDSTART = FALSE
LDAT_ACT = LCPDAT2987
FDAT_ACT = FP2987
BAS(#CP_PARAMS, 2.0)
SET_CD_PARAMS (0)
LIN XP2987
;ENDFOLD

;FOLD LIN P2988 Vel=2 m/s CPDAT2988 Tool[1]:marker Base[0] ;%{PE}
;FOLD Parameters ;%{h}
;Params IlfProvider=kukaroboter.basistech.inlineforms.movement.old; Kuka.IsGlobalPoint=False; Kuka.PointName=P2988; Kuka.BlendingEnabled=False; Kuka.MoveDataName=CPDAT1; Kuka.VelocityPath=2; Kuka.CurrentCDSetIndex=0; Kuka.MovementParameterFieldEnabled=True; IlfCommand=LIN
;ENDFOLD
$BWDSTART = FALSE
LDAT_ACT = LCPDAT2988
FDAT_ACT = FP2988
BAS(#CP_PARAMS, 2.0)
SET_CD_PARAMS (0)
LIN XP2988
;ENDFOLD

;FOLD LIN P2989 Vel=2 m/s CPDAT2989 Tool[1]:marker Base[0] ;%{PE}
;FOLD Parameters ;%{h}
;Params IlfProvider=kukaroboter.basistech.inlineforms.movement.old; Kuka.IsGlobalPoint=False; Kuka.PointName=P2989; Kuka.BlendingEnabled=False; Kuka.MoveDataName=CPDAT1; Kuka.VelocityPath=2; Kuka.CurrentCDSetIndex=0; Kuka.MovementParameterFieldEnabled=True; IlfCommand=LIN
;ENDFOLD
$BWDSTART = FALSE
LDAT_ACT = LCPDAT2989
FDAT_ACT = FP2989
BAS(#CP_PARAMS, 2.0)
SET_CD_PARAMS (0)
LIN XP2989
;ENDFOLD

;FOLD LIN P2990 Vel=2 m/s CPDAT2990 Tool[1]:marker Base[0] ;%{PE}
;FOLD Parameters ;%{h}
;Params IlfProvider=kukaroboter.basistech.inlineforms.movement.old; Kuka.IsGlobalPoint=False; Kuka.PointName=P2990; Kuka.BlendingEnabled=False; Kuka.MoveDataName=CPDAT1; Kuka.VelocityPath=2; Kuka.CurrentCDSetIndex=0; Kuka.MovementParameterFieldEnabled=True; IlfCommand=LIN
;ENDFOLD
$BWDSTART = FALSE
LDAT_ACT = LCPDAT2990
FDAT_ACT = FP2990
BAS(#CP_PARAMS, 2.0)
SET_CD_PARAMS (0)
LIN XP2990
;ENDFOLD

;FOLD LIN P2991 Vel=2 m/s CPDAT2991 Tool[1]:marker Base[0] ;%{PE}
;FOLD Parameters ;%{h}
;Params IlfProvider=kukaroboter.basistech.inlineforms.movement.old; Kuka.IsGlobalPoint=False; Kuka.PointName=P2991; Kuka.BlendingEnabled=False; Kuka.MoveDataName=CPDAT1; Kuka.VelocityPath=2; Kuka.CurrentCDSetIndex=0; Kuka.MovementParameterFieldEnabled=True; IlfCommand=LIN
;ENDFOLD
$BWDSTART = FALSE
LDAT_ACT = LCPDAT2991
FDAT_ACT = FP2991
BAS(#CP_PARAMS, 2.0)
SET_CD_PARAMS (0)
LIN XP2991
;ENDFOLD

;FOLD LIN P2992 Vel=2 m/s CPDAT2992 Tool[1]:marker Base[0] ;%{PE}
;FOLD Parameters ;%{h}
;Params IlfProvider=kukaroboter.basistech.inlineforms.movement.old; Kuka.IsGlobalPoint=False; Kuka.PointName=P2992; Kuka.BlendingEnabled=False; Kuka.MoveDataName=CPDAT1; Kuka.VelocityPath=2; Kuka.CurrentCDSetIndex=0; Kuka.MovementParameterFieldEnabled=True; IlfCommand=LIN
;ENDFOLD
$BWDSTART = FALSE
LDAT_ACT = LCPDAT2992
FDAT_ACT = FP2992
BAS(#CP_PARAMS, 2.0)
SET_CD_PARAMS (0)
LIN XP2992
;ENDFOLD

;FOLD LIN P2993 Vel=2 m/s CPDAT2993 Tool[1]:marker Base[0] ;%{PE}
;FOLD Parameters ;%{h}
;Params IlfProvider=kukaroboter.basistech.inlineforms.movement.old; Kuka.IsGlobalPoint=False; Kuka.PointName=P2993; Kuka.BlendingEnabled=False; Kuka.MoveDataName=CPDAT1; Kuka.VelocityPath=2; Kuka.CurrentCDSetIndex=0; Kuka.MovementParameterFieldEnabled=True; IlfCommand=LIN
;ENDFOLD
$BWDSTART = FALSE
LDAT_ACT = LCPDAT2993
FDAT_ACT = FP2993
BAS(#CP_PARAMS, 2.0)
SET_CD_PARAMS (0)
LIN XP2993
;ENDFOLD

;FOLD LIN P2994 Vel=2 m/s CPDAT2994 Tool[1]:marker Base[0] ;%{PE}
;FOLD Parameters ;%{h}
;Params IlfProvider=kukaroboter.basistech.inlineforms.movement.old; Kuka.IsGlobalPoint=False; Kuka.PointName=P2994; Kuka.BlendingEnabled=False; Kuka.MoveDataName=CPDAT1; Kuka.VelocityPath=2; Kuka.CurrentCDSetIndex=0; Kuka.MovementParameterFieldEnabled=True; IlfCommand=LIN
;ENDFOLD
$BWDSTART = FALSE
LDAT_ACT = LCPDAT2994
FDAT_ACT = FP2994
BAS(#CP_PARAMS, 2.0)
SET_CD_PARAMS (0)
LIN XP2994
;ENDFOLD

;FOLD LIN P2995 Vel=2 m/s CPDAT2995 Tool[1]:marker Base[0] ;%{PE}
;FOLD Parameters ;%{h}
;Params IlfProvider=kukaroboter.basistech.inlineforms.movement.old; Kuka.IsGlobalPoint=False; Kuka.PointName=P2995; Kuka.BlendingEnabled=False; Kuka.MoveDataName=CPDAT1; Kuka.VelocityPath=2; Kuka.CurrentCDSetIndex=0; Kuka.MovementParameterFieldEnabled=True; IlfCommand=LIN
;ENDFOLD
$BWDSTART = FALSE
LDAT_ACT = LCPDAT2995
FDAT_ACT = FP2995
BAS(#CP_PARAMS, 2.0)
SET_CD_PARAMS (0)
LIN XP2995
;ENDFOLD

;FOLD LIN P2996 Vel=2 m/s CPDAT2996 Tool[1]:marker Base[0] ;%{PE}
;FOLD Parameters ;%{h}
;Params IlfProvider=kukaroboter.basistech.inlineforms.movement.old; Kuka.IsGlobalPoint=False; Kuka.PointName=P2996; Kuka.BlendingEnabled=False; Kuka.MoveDataName=CPDAT1; Kuka.VelocityPath=2; Kuka.CurrentCDSetIndex=0; Kuka.MovementParameterFieldEnabled=True; IlfCommand=LIN
;ENDFOLD
$BWDSTART = FALSE
LDAT_ACT = LCPDAT2996
FDAT_ACT = FP2996
BAS(#CP_PARAMS, 2.0)
SET_CD_PARAMS (0)
LIN XP2996
;ENDFOLD

;FOLD LIN P2997 Vel=2 m/s CPDAT2997 Tool[1]:marker Base[0] ;%{PE}
;FOLD Parameters ;%{h}
;Params IlfProvider=kukaroboter.basistech.inlineforms.movement.old; Kuka.IsGlobalPoint=False; Kuka.PointName=P2997; Kuka.BlendingEnabled=False; Kuka.MoveDataName=CPDAT1; Kuka.VelocityPath=2; Kuka.CurrentCDSetIndex=0; Kuka.MovementParameterFieldEnabled=True; IlfCommand=LIN
;ENDFOLD
$BWDSTART = FALSE
LDAT_ACT = LCPDAT2997
FDAT_ACT = FP2997
BAS(#CP_PARAMS, 2.0)
SET_CD_PARAMS (0)
LIN XP2997
;ENDFOLD

;FOLD LIN P2998 Vel=2 m/s CPDAT2998 Tool[1]:marker Base[0] ;%{PE}
;FOLD Parameters ;%{h}
;Params IlfProvider=kukaroboter.basistech.inlineforms.movement.old; Kuka.IsGlobalPoint=False; Kuka.PointName=P2998; Kuka.BlendingEnabled=False; Kuka.MoveDataName=CPDAT1; Kuka.VelocityPath=2; Kuka.CurrentCDSetIndex=0; Kuka.MovementParameterFieldEnabled=True; IlfCommand=LIN
;ENDFOLD
$BWDSTART = FALSE
LDAT_ACT = LCPDAT2998
FDAT_ACT = FP2998
BAS(#CP_PARAMS, 2.0)
SET_CD_PARAMS (0)
LIN XP2998
;ENDFOLD

;FOLD LIN P2999 Vel=2 m/s CPDAT2999 Tool[1]:marker Base[0] ;%{PE}
;FOLD Parameters ;%{h}
;Params IlfProvider=kukaroboter.basistech.inlineforms.movement.old; Kuka.IsGlobalPoint=False; Kuka.PointName=P2999; Kuka.BlendingEnabled=False; Kuka.MoveDataName=CPDAT1; Kuka.VelocityPath=2; Kuka.CurrentCDSetIndex=0; Kuka.MovementParameterFieldEnabled=True; IlfCommand=LIN
;ENDFOLD
$BWDSTART = FALSE
LDAT_ACT = LCPDAT2999
FDAT_ACT = FP2999
BAS(#CP_PARAMS, 2.0)
SET_CD_PARAMS (0)
LIN XP2999
;ENDFOLD

;FOLD LIN P3000 Vel=2 m/s CPDAT3000 Tool[1]:marker Base[0] ;%{PE}
;FOLD Parameters ;%{h}
;Params IlfProvider=kukaroboter.basistech.inlineforms.movement.old; Kuka.IsGlobalPoint=False; Kuka.PointName=P3000; Kuka.BlendingEnabled=False; Kuka.MoveDataName=CPDAT1; Kuka.VelocityPath=2; Kuka.CurrentCDSetIndex=0; Kuka.MovementParameterFieldEnabled=True; IlfCommand=LIN
;ENDFOLD
$BWDSTART = FALSE
LDAT_ACT = LCPDAT3000
FDAT_ACT = FP3000
BAS(#CP_PARAMS, 2.0)
SET_CD_PARAMS (0)
LIN XP3000
;ENDFOLD

;FOLD LIN P3001 Vel=2 m/s CPDAT3001 Tool[1]:marker Base[0] ;%{PE}
;FOLD Parameters ;%{h}
;Params IlfProvider=kukaroboter.basistech.inlineforms.movement.old; Kuka.IsGlobalPoint=False; Kuka.PointName=P3001; Kuka.BlendingEnabled=False; Kuka.MoveDataName=CPDAT1; Kuka.VelocityPath=2; Kuka.CurrentCDSetIndex=0; Kuka.MovementParameterFieldEnabled=True; IlfCommand=LIN
;ENDFOLD
$BWDSTART = FALSE
LDAT_ACT = LCPDAT3001
FDAT_ACT = FP3001
BAS(#CP_PARAMS, 2.0)
SET_CD_PARAMS (0)
LIN XP3001
;ENDFOLD

;FOLD LIN P3002 Vel=2 m/s CPDAT3002 Tool[1]:marker Base[0] ;%{PE}
;FOLD Parameters ;%{h}
;Params IlfProvider=kukaroboter.basistech.inlineforms.movement.old; Kuka.IsGlobalPoint=False; Kuka.PointName=P3002; Kuka.BlendingEnabled=False; Kuka.MoveDataName=CPDAT1; Kuka.VelocityPath=2; Kuka.CurrentCDSetIndex=0; Kuka.MovementParameterFieldEnabled=True; IlfCommand=LIN
;ENDFOLD
$BWDSTART = FALSE
LDAT_ACT = LCPDAT3002
FDAT_ACT = FP3002
BAS(#CP_PARAMS, 2.0)
SET_CD_PARAMS (0)
LIN XP3002
;ENDFOLD

;FOLD LIN P3003 Vel=2 m/s CPDAT3003 Tool[1]:marker Base[0] ;%{PE}
;FOLD Parameters ;%{h}
;Params IlfProvider=kukaroboter.basistech.inlineforms.movement.old; Kuka.IsGlobalPoint=False; Kuka.PointName=P3003; Kuka.BlendingEnabled=False; Kuka.MoveDataName=CPDAT1; Kuka.VelocityPath=2; Kuka.CurrentCDSetIndex=0; Kuka.MovementParameterFieldEnabled=True; IlfCommand=LIN
;ENDFOLD
$BWDSTART = FALSE
LDAT_ACT = LCPDAT3003
FDAT_ACT = FP3003
BAS(#CP_PARAMS, 2.0)
SET_CD_PARAMS (0)
LIN XP3003
;ENDFOLD

;FOLD LIN P3004 Vel=2 m/s CPDAT3004 Tool[1]:marker Base[0] ;%{PE}
;FOLD Parameters ;%{h}
;Params IlfProvider=kukaroboter.basistech.inlineforms.movement.old; Kuka.IsGlobalPoint=False; Kuka.PointName=P3004; Kuka.BlendingEnabled=False; Kuka.MoveDataName=CPDAT1; Kuka.VelocityPath=2; Kuka.CurrentCDSetIndex=0; Kuka.MovementParameterFieldEnabled=True; IlfCommand=LIN
;ENDFOLD
$BWDSTART = FALSE
LDAT_ACT = LCPDAT3004
FDAT_ACT = FP3004
BAS(#CP_PARAMS, 2.0)
SET_CD_PARAMS (0)
LIN XP3004
;ENDFOLD

;FOLD LIN P3005 Vel=2 m/s CPDAT3005 Tool[1]:marker Base[0] ;%{PE}
;FOLD Parameters ;%{h}
;Params IlfProvider=kukaroboter.basistech.inlineforms.movement.old; Kuka.IsGlobalPoint=False; Kuka.PointName=P3005; Kuka.BlendingEnabled=False; Kuka.MoveDataName=CPDAT1; Kuka.VelocityPath=2; Kuka.CurrentCDSetIndex=0; Kuka.MovementParameterFieldEnabled=True; IlfCommand=LIN
;ENDFOLD
$BWDSTART = FALSE
LDAT_ACT = LCPDAT3005
FDAT_ACT = FP3005
BAS(#CP_PARAMS, 2.0)
SET_CD_PARAMS (0)
LIN XP3005
;ENDFOLD

;FOLD LIN P3006 Vel=2 m/s CPDAT3006 Tool[1]:marker Base[0] ;%{PE}
;FOLD Parameters ;%{h}
;Params IlfProvider=kukaroboter.basistech.inlineforms.movement.old; Kuka.IsGlobalPoint=False; Kuka.PointName=P3006; Kuka.BlendingEnabled=False; Kuka.MoveDataName=CPDAT1; Kuka.VelocityPath=2; Kuka.CurrentCDSetIndex=0; Kuka.MovementParameterFieldEnabled=True; IlfCommand=LIN
;ENDFOLD
$BWDSTART = FALSE
LDAT_ACT = LCPDAT3006
FDAT_ACT = FP3006
BAS(#CP_PARAMS, 2.0)
SET_CD_PARAMS (0)
LIN XP3006
;ENDFOLD

;FOLD LIN P3007 Vel=2 m/s CPDAT3007 Tool[1]:marker Base[0] ;%{PE}
;FOLD Parameters ;%{h}
;Params IlfProvider=kukaroboter.basistech.inlineforms.movement.old; Kuka.IsGlobalPoint=False; Kuka.PointName=P3007; Kuka.BlendingEnabled=False; Kuka.MoveDataName=CPDAT1; Kuka.VelocityPath=2; Kuka.CurrentCDSetIndex=0; Kuka.MovementParameterFieldEnabled=True; IlfCommand=LIN
;ENDFOLD
$BWDSTART = FALSE
LDAT_ACT = LCPDAT3007
FDAT_ACT = FP3007
BAS(#CP_PARAMS, 2.0)
SET_CD_PARAMS (0)
LIN XP3007
;ENDFOLD

;FOLD LIN P3008 Vel=2 m/s CPDAT3008 Tool[1]:marker Base[0] ;%{PE}
;FOLD Parameters ;%{h}
;Params IlfProvider=kukaroboter.basistech.inlineforms.movement.old; Kuka.IsGlobalPoint=False; Kuka.PointName=P3008; Kuka.BlendingEnabled=False; Kuka.MoveDataName=CPDAT1; Kuka.VelocityPath=2; Kuka.CurrentCDSetIndex=0; Kuka.MovementParameterFieldEnabled=True; IlfCommand=LIN
;ENDFOLD
$BWDSTART = FALSE
LDAT_ACT = LCPDAT3008
FDAT_ACT = FP3008
BAS(#CP_PARAMS, 2.0)
SET_CD_PARAMS (0)
LIN XP3008
;ENDFOLD

;FOLD LIN P3009 Vel=2 m/s CPDAT3009 Tool[1]:marker Base[0] ;%{PE}
;FOLD Parameters ;%{h}
;Params IlfProvider=kukaroboter.basistech.inlineforms.movement.old; Kuka.IsGlobalPoint=False; Kuka.PointName=P3009; Kuka.BlendingEnabled=False; Kuka.MoveDataName=CPDAT1; Kuka.VelocityPath=2; Kuka.CurrentCDSetIndex=0; Kuka.MovementParameterFieldEnabled=True; IlfCommand=LIN
;ENDFOLD
$BWDSTART = FALSE
LDAT_ACT = LCPDAT3009
FDAT_ACT = FP3009
BAS(#CP_PARAMS, 2.0)
SET_CD_PARAMS (0)
LIN XP3009
;ENDFOLD

;FOLD LIN P3010 Vel=2 m/s CPDAT3010 Tool[1]:marker Base[0] ;%{PE}
;FOLD Parameters ;%{h}
;Params IlfProvider=kukaroboter.basistech.inlineforms.movement.old; Kuka.IsGlobalPoint=False; Kuka.PointName=P3010; Kuka.BlendingEnabled=False; Kuka.MoveDataName=CPDAT1; Kuka.VelocityPath=2; Kuka.CurrentCDSetIndex=0; Kuka.MovementParameterFieldEnabled=True; IlfCommand=LIN
;ENDFOLD
$BWDSTART = FALSE
LDAT_ACT = LCPDAT3010
FDAT_ACT = FP3010
BAS(#CP_PARAMS, 2.0)
SET_CD_PARAMS (0)
LIN XP3010
;ENDFOLD

;FOLD LIN P3011 Vel=2 m/s CPDAT3011 Tool[1]:marker Base[0] ;%{PE}
;FOLD Parameters ;%{h}
;Params IlfProvider=kukaroboter.basistech.inlineforms.movement.old; Kuka.IsGlobalPoint=False; Kuka.PointName=P3011; Kuka.BlendingEnabled=False; Kuka.MoveDataName=CPDAT1; Kuka.VelocityPath=2; Kuka.CurrentCDSetIndex=0; Kuka.MovementParameterFieldEnabled=True; IlfCommand=LIN
;ENDFOLD
$BWDSTART = FALSE
LDAT_ACT = LCPDAT3011
FDAT_ACT = FP3011
BAS(#CP_PARAMS, 2.0)
SET_CD_PARAMS (0)
LIN XP3011
;ENDFOLD

;FOLD LIN P3012 Vel=2 m/s CPDAT3012 Tool[1]:marker Base[0] ;%{PE}
;FOLD Parameters ;%{h}
;Params IlfProvider=kukaroboter.basistech.inlineforms.movement.old; Kuka.IsGlobalPoint=False; Kuka.PointName=P3012; Kuka.BlendingEnabled=False; Kuka.MoveDataName=CPDAT1; Kuka.VelocityPath=2; Kuka.CurrentCDSetIndex=0; Kuka.MovementParameterFieldEnabled=True; IlfCommand=LIN
;ENDFOLD
$BWDSTART = FALSE
LDAT_ACT = LCPDAT3012
FDAT_ACT = FP3012
BAS(#CP_PARAMS, 2.0)
SET_CD_PARAMS (0)
LIN XP3012
;ENDFOLD

;FOLD LIN P3013 Vel=2 m/s CPDAT3013 Tool[1]:marker Base[0] ;%{PE}
;FOLD Parameters ;%{h}
;Params IlfProvider=kukaroboter.basistech.inlineforms.movement.old; Kuka.IsGlobalPoint=False; Kuka.PointName=P3013; Kuka.BlendingEnabled=False; Kuka.MoveDataName=CPDAT1; Kuka.VelocityPath=2; Kuka.CurrentCDSetIndex=0; Kuka.MovementParameterFieldEnabled=True; IlfCommand=LIN
;ENDFOLD
$BWDSTART = FALSE
LDAT_ACT = LCPDAT3013
FDAT_ACT = FP3013
BAS(#CP_PARAMS, 2.0)
SET_CD_PARAMS (0)
LIN XP3013
;ENDFOLD

;FOLD LIN P3014 Vel=2 m/s CPDAT3014 Tool[1]:marker Base[0] ;%{PE}
;FOLD Parameters ;%{h}
;Params IlfProvider=kukaroboter.basistech.inlineforms.movement.old; Kuka.IsGlobalPoint=False; Kuka.PointName=P3014; Kuka.BlendingEnabled=False; Kuka.MoveDataName=CPDAT1; Kuka.VelocityPath=2; Kuka.CurrentCDSetIndex=0; Kuka.MovementParameterFieldEnabled=True; IlfCommand=LIN
;ENDFOLD
$BWDSTART = FALSE
LDAT_ACT = LCPDAT3014
FDAT_ACT = FP3014
BAS(#CP_PARAMS, 2.0)
SET_CD_PARAMS (0)
LIN XP3014
;ENDFOLD

;FOLD LIN P3015 Vel=2 m/s CPDAT3015 Tool[1]:marker Base[0] ;%{PE}
;FOLD Parameters ;%{h}
;Params IlfProvider=kukaroboter.basistech.inlineforms.movement.old; Kuka.IsGlobalPoint=False; Kuka.PointName=P3015; Kuka.BlendingEnabled=False; Kuka.MoveDataName=CPDAT1; Kuka.VelocityPath=2; Kuka.CurrentCDSetIndex=0; Kuka.MovementParameterFieldEnabled=True; IlfCommand=LIN
;ENDFOLD
$BWDSTART = FALSE
LDAT_ACT = LCPDAT3015
FDAT_ACT = FP3015
BAS(#CP_PARAMS, 2.0)
SET_CD_PARAMS (0)
LIN XP3015
;ENDFOLD

;FOLD LIN P3016 Vel=2 m/s CPDAT3016 Tool[1]:marker Base[0] ;%{PE}
;FOLD Parameters ;%{h}
;Params IlfProvider=kukaroboter.basistech.inlineforms.movement.old; Kuka.IsGlobalPoint=False; Kuka.PointName=P3016; Kuka.BlendingEnabled=False; Kuka.MoveDataName=CPDAT1; Kuka.VelocityPath=2; Kuka.CurrentCDSetIndex=0; Kuka.MovementParameterFieldEnabled=True; IlfCommand=LIN
;ENDFOLD
$BWDSTART = FALSE
LDAT_ACT = LCPDAT3016
FDAT_ACT = FP3016
BAS(#CP_PARAMS, 2.0)
SET_CD_PARAMS (0)
LIN XP3016
;ENDFOLD

;FOLD LIN P3017 Vel=2 m/s CPDAT3017 Tool[1]:marker Base[0] ;%{PE}
;FOLD Parameters ;%{h}
;Params IlfProvider=kukaroboter.basistech.inlineforms.movement.old; Kuka.IsGlobalPoint=False; Kuka.PointName=P3017; Kuka.BlendingEnabled=False; Kuka.MoveDataName=CPDAT1; Kuka.VelocityPath=2; Kuka.CurrentCDSetIndex=0; Kuka.MovementParameterFieldEnabled=True; IlfCommand=LIN
;ENDFOLD
$BWDSTART = FALSE
LDAT_ACT = LCPDAT3017
FDAT_ACT = FP3017
BAS(#CP_PARAMS, 2.0)
SET_CD_PARAMS (0)
LIN XP3017
;ENDFOLD

;FOLD LIN P3018 Vel=2 m/s CPDAT3018 Tool[1]:marker Base[0] ;%{PE}
;FOLD Parameters ;%{h}
;Params IlfProvider=kukaroboter.basistech.inlineforms.movement.old; Kuka.IsGlobalPoint=False; Kuka.PointName=P3018; Kuka.BlendingEnabled=False; Kuka.MoveDataName=CPDAT1; Kuka.VelocityPath=2; Kuka.CurrentCDSetIndex=0; Kuka.MovementParameterFieldEnabled=True; IlfCommand=LIN
;ENDFOLD
$BWDSTART = FALSE
LDAT_ACT = LCPDAT3018
FDAT_ACT = FP3018
BAS(#CP_PARAMS, 2.0)
SET_CD_PARAMS (0)
LIN XP3018
;ENDFOLD

;FOLD LIN P3019 Vel=2 m/s CPDAT3019 Tool[1]:marker Base[0] ;%{PE}
;FOLD Parameters ;%{h}
;Params IlfProvider=kukaroboter.basistech.inlineforms.movement.old; Kuka.IsGlobalPoint=False; Kuka.PointName=P3019; Kuka.BlendingEnabled=False; Kuka.MoveDataName=CPDAT1; Kuka.VelocityPath=2; Kuka.CurrentCDSetIndex=0; Kuka.MovementParameterFieldEnabled=True; IlfCommand=LIN
;ENDFOLD
$BWDSTART = FALSE
LDAT_ACT = LCPDAT3019
FDAT_ACT = FP3019
BAS(#CP_PARAMS, 2.0)
SET_CD_PARAMS (0)
LIN XP3019
;ENDFOLD

;FOLD LIN P3020 Vel=2 m/s CPDAT3020 Tool[1]:marker Base[0] ;%{PE}
;FOLD Parameters ;%{h}
;Params IlfProvider=kukaroboter.basistech.inlineforms.movement.old; Kuka.IsGlobalPoint=False; Kuka.PointName=P3020; Kuka.BlendingEnabled=False; Kuka.MoveDataName=CPDAT1; Kuka.VelocityPath=2; Kuka.CurrentCDSetIndex=0; Kuka.MovementParameterFieldEnabled=True; IlfCommand=LIN
;ENDFOLD
$BWDSTART = FALSE
LDAT_ACT = LCPDAT3020
FDAT_ACT = FP3020
BAS(#CP_PARAMS, 2.0)
SET_CD_PARAMS (0)
LIN XP3020
;ENDFOLD

;FOLD LIN P3021 Vel=2 m/s CPDAT3021 Tool[1]:marker Base[0] ;%{PE}
;FOLD Parameters ;%{h}
;Params IlfProvider=kukaroboter.basistech.inlineforms.movement.old; Kuka.IsGlobalPoint=False; Kuka.PointName=P3021; Kuka.BlendingEnabled=False; Kuka.MoveDataName=CPDAT1; Kuka.VelocityPath=2; Kuka.CurrentCDSetIndex=0; Kuka.MovementParameterFieldEnabled=True; IlfCommand=LIN
;ENDFOLD
$BWDSTART = FALSE
LDAT_ACT = LCPDAT3021
FDAT_ACT = FP3021
BAS(#CP_PARAMS, 2.0)
SET_CD_PARAMS (0)
LIN XP3021
;ENDFOLD

;FOLD LIN P3022 Vel=2 m/s CPDAT3022 Tool[1]:marker Base[0] ;%{PE}
;FOLD Parameters ;%{h}
;Params IlfProvider=kukaroboter.basistech.inlineforms.movement.old; Kuka.IsGlobalPoint=False; Kuka.PointName=P3022; Kuka.BlendingEnabled=False; Kuka.MoveDataName=CPDAT1; Kuka.VelocityPath=2; Kuka.CurrentCDSetIndex=0; Kuka.MovementParameterFieldEnabled=True; IlfCommand=LIN
;ENDFOLD
$BWDSTART = FALSE
LDAT_ACT = LCPDAT3022
FDAT_ACT = FP3022
BAS(#CP_PARAMS, 2.0)
SET_CD_PARAMS (0)
LIN XP3022
;ENDFOLD

;FOLD LIN P3023 Vel=2 m/s CPDAT3023 Tool[1]:marker Base[0] ;%{PE}
;FOLD Parameters ;%{h}
;Params IlfProvider=kukaroboter.basistech.inlineforms.movement.old; Kuka.IsGlobalPoint=False; Kuka.PointName=P3023; Kuka.BlendingEnabled=False; Kuka.MoveDataName=CPDAT1; Kuka.VelocityPath=2; Kuka.CurrentCDSetIndex=0; Kuka.MovementParameterFieldEnabled=True; IlfCommand=LIN
;ENDFOLD
$BWDSTART = FALSE
LDAT_ACT = LCPDAT3023
FDAT_ACT = FP3023
BAS(#CP_PARAMS, 2.0)
SET_CD_PARAMS (0)
LIN XP3023
;ENDFOLD

;FOLD LIN P3024 Vel=2 m/s CPDAT3024 Tool[1]:marker Base[0] ;%{PE}
;FOLD Parameters ;%{h}
;Params IlfProvider=kukaroboter.basistech.inlineforms.movement.old; Kuka.IsGlobalPoint=False; Kuka.PointName=P3024; Kuka.BlendingEnabled=False; Kuka.MoveDataName=CPDAT1; Kuka.VelocityPath=2; Kuka.CurrentCDSetIndex=0; Kuka.MovementParameterFieldEnabled=True; IlfCommand=LIN
;ENDFOLD
$BWDSTART = FALSE
LDAT_ACT = LCPDAT3024
FDAT_ACT = FP3024
BAS(#CP_PARAMS, 2.0)
SET_CD_PARAMS (0)
LIN XP3024
;ENDFOLD

;FOLD LIN P3025 Vel=2 m/s CPDAT3025 Tool[1]:marker Base[0] ;%{PE}
;FOLD Parameters ;%{h}
;Params IlfProvider=kukaroboter.basistech.inlineforms.movement.old; Kuka.IsGlobalPoint=False; Kuka.PointName=P3025; Kuka.BlendingEnabled=False; Kuka.MoveDataName=CPDAT1; Kuka.VelocityPath=2; Kuka.CurrentCDSetIndex=0; Kuka.MovementParameterFieldEnabled=True; IlfCommand=LIN
;ENDFOLD
$BWDSTART = FALSE
LDAT_ACT = LCPDAT3025
FDAT_ACT = FP3025
BAS(#CP_PARAMS, 2.0)
SET_CD_PARAMS (0)
LIN XP3025
;ENDFOLD

;FOLD LIN P3026 Vel=2 m/s CPDAT3026 Tool[1]:marker Base[0] ;%{PE}
;FOLD Parameters ;%{h}
;Params IlfProvider=kukaroboter.basistech.inlineforms.movement.old; Kuka.IsGlobalPoint=False; Kuka.PointName=P3026; Kuka.BlendingEnabled=False; Kuka.MoveDataName=CPDAT1; Kuka.VelocityPath=2; Kuka.CurrentCDSetIndex=0; Kuka.MovementParameterFieldEnabled=True; IlfCommand=LIN
;ENDFOLD
$BWDSTART = FALSE
LDAT_ACT = LCPDAT3026
FDAT_ACT = FP3026
BAS(#CP_PARAMS, 2.0)
SET_CD_PARAMS (0)
LIN XP3026
;ENDFOLD

;FOLD LIN P3027 Vel=2 m/s CPDAT3027 Tool[1]:marker Base[0] ;%{PE}
;FOLD Parameters ;%{h}
;Params IlfProvider=kukaroboter.basistech.inlineforms.movement.old; Kuka.IsGlobalPoint=False; Kuka.PointName=P3027; Kuka.BlendingEnabled=False; Kuka.MoveDataName=CPDAT1; Kuka.VelocityPath=2; Kuka.CurrentCDSetIndex=0; Kuka.MovementParameterFieldEnabled=True; IlfCommand=LIN
;ENDFOLD
$BWDSTART = FALSE
LDAT_ACT = LCPDAT3027
FDAT_ACT = FP3027
BAS(#CP_PARAMS, 2.0)
SET_CD_PARAMS (0)
LIN XP3027
;ENDFOLD

;FOLD LIN P3028 Vel=2 m/s CPDAT3028 Tool[1]:marker Base[0] ;%{PE}
;FOLD Parameters ;%{h}
;Params IlfProvider=kukaroboter.basistech.inlineforms.movement.old; Kuka.IsGlobalPoint=False; Kuka.PointName=P3028; Kuka.BlendingEnabled=False; Kuka.MoveDataName=CPDAT1; Kuka.VelocityPath=2; Kuka.CurrentCDSetIndex=0; Kuka.MovementParameterFieldEnabled=True; IlfCommand=LIN
;ENDFOLD
$BWDSTART = FALSE
LDAT_ACT = LCPDAT3028
FDAT_ACT = FP3028
BAS(#CP_PARAMS, 2.0)
SET_CD_PARAMS (0)
LIN XP3028
;ENDFOLD

;FOLD LIN P3029 Vel=2 m/s CPDAT3029 Tool[1]:marker Base[0] ;%{PE}
;FOLD Parameters ;%{h}
;Params IlfProvider=kukaroboter.basistech.inlineforms.movement.old; Kuka.IsGlobalPoint=False; Kuka.PointName=P3029; Kuka.BlendingEnabled=False; Kuka.MoveDataName=CPDAT1; Kuka.VelocityPath=2; Kuka.CurrentCDSetIndex=0; Kuka.MovementParameterFieldEnabled=True; IlfCommand=LIN
;ENDFOLD
$BWDSTART = FALSE
LDAT_ACT = LCPDAT3029
FDAT_ACT = FP3029
BAS(#CP_PARAMS, 2.0)
SET_CD_PARAMS (0)
LIN XP3029
;ENDFOLD

;FOLD LIN P3030 Vel=2 m/s CPDAT3030 Tool[1]:marker Base[0] ;%{PE}
;FOLD Parameters ;%{h}
;Params IlfProvider=kukaroboter.basistech.inlineforms.movement.old; Kuka.IsGlobalPoint=False; Kuka.PointName=P3030; Kuka.BlendingEnabled=False; Kuka.MoveDataName=CPDAT1; Kuka.VelocityPath=2; Kuka.CurrentCDSetIndex=0; Kuka.MovementParameterFieldEnabled=True; IlfCommand=LIN
;ENDFOLD
$BWDSTART = FALSE
LDAT_ACT = LCPDAT3030
FDAT_ACT = FP3030
BAS(#CP_PARAMS, 2.0)
SET_CD_PARAMS (0)
LIN XP3030
;ENDFOLD

;FOLD LIN P3031 Vel=2 m/s CPDAT3031 Tool[1]:marker Base[0] ;%{PE}
;FOLD Parameters ;%{h}
;Params IlfProvider=kukaroboter.basistech.inlineforms.movement.old; Kuka.IsGlobalPoint=False; Kuka.PointName=P3031; Kuka.BlendingEnabled=False; Kuka.MoveDataName=CPDAT1; Kuka.VelocityPath=2; Kuka.CurrentCDSetIndex=0; Kuka.MovementParameterFieldEnabled=True; IlfCommand=LIN
;ENDFOLD
$BWDSTART = FALSE
LDAT_ACT = LCPDAT3031
FDAT_ACT = FP3031
BAS(#CP_PARAMS, 2.0)
SET_CD_PARAMS (0)
LIN XP3031
;ENDFOLD

;FOLD LIN P3032 Vel=2 m/s CPDAT3032 Tool[1]:marker Base[0] ;%{PE}
;FOLD Parameters ;%{h}
;Params IlfProvider=kukaroboter.basistech.inlineforms.movement.old; Kuka.IsGlobalPoint=False; Kuka.PointName=P3032; Kuka.BlendingEnabled=False; Kuka.MoveDataName=CPDAT1; Kuka.VelocityPath=2; Kuka.CurrentCDSetIndex=0; Kuka.MovementParameterFieldEnabled=True; IlfCommand=LIN
;ENDFOLD
$BWDSTART = FALSE
LDAT_ACT = LCPDAT3032
FDAT_ACT = FP3032
BAS(#CP_PARAMS, 2.0)
SET_CD_PARAMS (0)
LIN XP3032
;ENDFOLD

;FOLD LIN P3033 Vel=2 m/s CPDAT3033 Tool[1]:marker Base[0] ;%{PE}
;FOLD Parameters ;%{h}
;Params IlfProvider=kukaroboter.basistech.inlineforms.movement.old; Kuka.IsGlobalPoint=False; Kuka.PointName=P3033; Kuka.BlendingEnabled=False; Kuka.MoveDataName=CPDAT1; Kuka.VelocityPath=2; Kuka.CurrentCDSetIndex=0; Kuka.MovementParameterFieldEnabled=True; IlfCommand=LIN
;ENDFOLD
$BWDSTART = FALSE
LDAT_ACT = LCPDAT3033
FDAT_ACT = FP3033
BAS(#CP_PARAMS, 2.0)
SET_CD_PARAMS (0)
LIN XP3033
;ENDFOLD

;FOLD LIN P3034 Vel=2 m/s CPDAT3034 Tool[1]:marker Base[0] ;%{PE}
;FOLD Parameters ;%{h}
;Params IlfProvider=kukaroboter.basistech.inlineforms.movement.old; Kuka.IsGlobalPoint=False; Kuka.PointName=P3034; Kuka.BlendingEnabled=False; Kuka.MoveDataName=CPDAT1; Kuka.VelocityPath=2; Kuka.CurrentCDSetIndex=0; Kuka.MovementParameterFieldEnabled=True; IlfCommand=LIN
;ENDFOLD
$BWDSTART = FALSE
LDAT_ACT = LCPDAT3034
FDAT_ACT = FP3034
BAS(#CP_PARAMS, 2.0)
SET_CD_PARAMS (0)
LIN XP3034
;ENDFOLD

;FOLD LIN P3035 Vel=2 m/s CPDAT3035 Tool[1]:marker Base[0] ;%{PE}
;FOLD Parameters ;%{h}
;Params IlfProvider=kukaroboter.basistech.inlineforms.movement.old; Kuka.IsGlobalPoint=False; Kuka.PointName=P3035; Kuka.BlendingEnabled=False; Kuka.MoveDataName=CPDAT1; Kuka.VelocityPath=2; Kuka.CurrentCDSetIndex=0; Kuka.MovementParameterFieldEnabled=True; IlfCommand=LIN
;ENDFOLD
$BWDSTART = FALSE
LDAT_ACT = LCPDAT3035
FDAT_ACT = FP3035
BAS(#CP_PARAMS, 2.0)
SET_CD_PARAMS (0)
LIN XP3035
;ENDFOLD

;FOLD LIN P3036 Vel=2 m/s CPDAT3036 Tool[1]:marker Base[0] ;%{PE}
;FOLD Parameters ;%{h}
;Params IlfProvider=kukaroboter.basistech.inlineforms.movement.old; Kuka.IsGlobalPoint=False; Kuka.PointName=P3036; Kuka.BlendingEnabled=False; Kuka.MoveDataName=CPDAT1; Kuka.VelocityPath=2; Kuka.CurrentCDSetIndex=0; Kuka.MovementParameterFieldEnabled=True; IlfCommand=LIN
;ENDFOLD
$BWDSTART = FALSE
LDAT_ACT = LCPDAT3036
FDAT_ACT = FP3036
BAS(#CP_PARAMS, 2.0)
SET_CD_PARAMS (0)
LIN XP3036
;ENDFOLD

;FOLD LIN P3037 Vel=2 m/s CPDAT3037 Tool[1]:marker Base[0] ;%{PE}
;FOLD Parameters ;%{h}
;Params IlfProvider=kukaroboter.basistech.inlineforms.movement.old; Kuka.IsGlobalPoint=False; Kuka.PointName=P3037; Kuka.BlendingEnabled=False; Kuka.MoveDataName=CPDAT1; Kuka.VelocityPath=2; Kuka.CurrentCDSetIndex=0; Kuka.MovementParameterFieldEnabled=True; IlfCommand=LIN
;ENDFOLD
$BWDSTART = FALSE
LDAT_ACT = LCPDAT3037
FDAT_ACT = FP3037
BAS(#CP_PARAMS, 2.0)
SET_CD_PARAMS (0)
LIN XP3037
;ENDFOLD

;FOLD LIN P3038 Vel=2 m/s CPDAT3038 Tool[1]:marker Base[0] ;%{PE}
;FOLD Parameters ;%{h}
;Params IlfProvider=kukaroboter.basistech.inlineforms.movement.old; Kuka.IsGlobalPoint=False; Kuka.PointName=P3038; Kuka.BlendingEnabled=False; Kuka.MoveDataName=CPDAT1; Kuka.VelocityPath=2; Kuka.CurrentCDSetIndex=0; Kuka.MovementParameterFieldEnabled=True; IlfCommand=LIN
;ENDFOLD
$BWDSTART = FALSE
LDAT_ACT = LCPDAT3038
FDAT_ACT = FP3038
BAS(#CP_PARAMS, 2.0)
SET_CD_PARAMS (0)
LIN XP3038
;ENDFOLD

;FOLD LIN P3039 Vel=2 m/s CPDAT3039 Tool[1]:marker Base[0] ;%{PE}
;FOLD Parameters ;%{h}
;Params IlfProvider=kukaroboter.basistech.inlineforms.movement.old; Kuka.IsGlobalPoint=False; Kuka.PointName=P3039; Kuka.BlendingEnabled=False; Kuka.MoveDataName=CPDAT1; Kuka.VelocityPath=2; Kuka.CurrentCDSetIndex=0; Kuka.MovementParameterFieldEnabled=True; IlfCommand=LIN
;ENDFOLD
$BWDSTART = FALSE
LDAT_ACT = LCPDAT3039
FDAT_ACT = FP3039
BAS(#CP_PARAMS, 2.0)
SET_CD_PARAMS (0)
LIN XP3039
;ENDFOLD

;FOLD LIN P3040 Vel=2 m/s CPDAT3040 Tool[1]:marker Base[0] ;%{PE}
;FOLD Parameters ;%{h}
;Params IlfProvider=kukaroboter.basistech.inlineforms.movement.old; Kuka.IsGlobalPoint=False; Kuka.PointName=P3040; Kuka.BlendingEnabled=False; Kuka.MoveDataName=CPDAT1; Kuka.VelocityPath=2; Kuka.CurrentCDSetIndex=0; Kuka.MovementParameterFieldEnabled=True; IlfCommand=LIN
;ENDFOLD
$BWDSTART = FALSE
LDAT_ACT = LCPDAT3040
FDAT_ACT = FP3040
BAS(#CP_PARAMS, 2.0)
SET_CD_PARAMS (0)
LIN XP3040
;ENDFOLD

;FOLD LIN P3041 Vel=2 m/s CPDAT3041 Tool[1]:marker Base[0] ;%{PE}
;FOLD Parameters ;%{h}
;Params IlfProvider=kukaroboter.basistech.inlineforms.movement.old; Kuka.IsGlobalPoint=False; Kuka.PointName=P3041; Kuka.BlendingEnabled=False; Kuka.MoveDataName=CPDAT1; Kuka.VelocityPath=2; Kuka.CurrentCDSetIndex=0; Kuka.MovementParameterFieldEnabled=True; IlfCommand=LIN
;ENDFOLD
$BWDSTART = FALSE
LDAT_ACT = LCPDAT3041
FDAT_ACT = FP3041
BAS(#CP_PARAMS, 2.0)
SET_CD_PARAMS (0)
LIN XP3041
;ENDFOLD

;FOLD LIN P3042 Vel=2 m/s CPDAT3042 Tool[1]:marker Base[0] ;%{PE}
;FOLD Parameters ;%{h}
;Params IlfProvider=kukaroboter.basistech.inlineforms.movement.old; Kuka.IsGlobalPoint=False; Kuka.PointName=P3042; Kuka.BlendingEnabled=False; Kuka.MoveDataName=CPDAT1; Kuka.VelocityPath=2; Kuka.CurrentCDSetIndex=0; Kuka.MovementParameterFieldEnabled=True; IlfCommand=LIN
;ENDFOLD
$BWDSTART = FALSE
LDAT_ACT = LCPDAT3042
FDAT_ACT = FP3042
BAS(#CP_PARAMS, 2.0)
SET_CD_PARAMS (0)
LIN XP3042
;ENDFOLD

;FOLD LIN P3043 Vel=2 m/s CPDAT3043 Tool[1]:marker Base[0] ;%{PE}
;FOLD Parameters ;%{h}
;Params IlfProvider=kukaroboter.basistech.inlineforms.movement.old; Kuka.IsGlobalPoint=False; Kuka.PointName=P3043; Kuka.BlendingEnabled=False; Kuka.MoveDataName=CPDAT1; Kuka.VelocityPath=2; Kuka.CurrentCDSetIndex=0; Kuka.MovementParameterFieldEnabled=True; IlfCommand=LIN
;ENDFOLD
$BWDSTART = FALSE
LDAT_ACT = LCPDAT3043
FDAT_ACT = FP3043
BAS(#CP_PARAMS, 2.0)
SET_CD_PARAMS (0)
LIN XP3043
;ENDFOLD

;FOLD LIN P3044 Vel=2 m/s CPDAT3044 Tool[1]:marker Base[0] ;%{PE}
;FOLD Parameters ;%{h}
;Params IlfProvider=kukaroboter.basistech.inlineforms.movement.old; Kuka.IsGlobalPoint=False; Kuka.PointName=P3044; Kuka.BlendingEnabled=False; Kuka.MoveDataName=CPDAT1; Kuka.VelocityPath=2; Kuka.CurrentCDSetIndex=0; Kuka.MovementParameterFieldEnabled=True; IlfCommand=LIN
;ENDFOLD
$BWDSTART = FALSE
LDAT_ACT = LCPDAT3044
FDAT_ACT = FP3044
BAS(#CP_PARAMS, 2.0)
SET_CD_PARAMS (0)
LIN XP3044
;ENDFOLD

;FOLD LIN P3045 Vel=2 m/s CPDAT3045 Tool[1]:marker Base[0] ;%{PE}
;FOLD Parameters ;%{h}
;Params IlfProvider=kukaroboter.basistech.inlineforms.movement.old; Kuka.IsGlobalPoint=False; Kuka.PointName=P3045; Kuka.BlendingEnabled=False; Kuka.MoveDataName=CPDAT1; Kuka.VelocityPath=2; Kuka.CurrentCDSetIndex=0; Kuka.MovementParameterFieldEnabled=True; IlfCommand=LIN
;ENDFOLD
$BWDSTART = FALSE
LDAT_ACT = LCPDAT3045
FDAT_ACT = FP3045
BAS(#CP_PARAMS, 2.0)
SET_CD_PARAMS (0)
LIN XP3045
;ENDFOLD

;FOLD LIN P3046 Vel=2 m/s CPDAT3046 Tool[1]:marker Base[0] ;%{PE}
;FOLD Parameters ;%{h}
;Params IlfProvider=kukaroboter.basistech.inlineforms.movement.old; Kuka.IsGlobalPoint=False; Kuka.PointName=P3046; Kuka.BlendingEnabled=False; Kuka.MoveDataName=CPDAT1; Kuka.VelocityPath=2; Kuka.CurrentCDSetIndex=0; Kuka.MovementParameterFieldEnabled=True; IlfCommand=LIN
;ENDFOLD
$BWDSTART = FALSE
LDAT_ACT = LCPDAT3046
FDAT_ACT = FP3046
BAS(#CP_PARAMS, 2.0)
SET_CD_PARAMS (0)
LIN XP3046
;ENDFOLD

;FOLD LIN P3047 Vel=2 m/s CPDAT3047 Tool[1]:marker Base[0] ;%{PE}
;FOLD Parameters ;%{h}
;Params IlfProvider=kukaroboter.basistech.inlineforms.movement.old; Kuka.IsGlobalPoint=False; Kuka.PointName=P3047; Kuka.BlendingEnabled=False; Kuka.MoveDataName=CPDAT1; Kuka.VelocityPath=2; Kuka.CurrentCDSetIndex=0; Kuka.MovementParameterFieldEnabled=True; IlfCommand=LIN
;ENDFOLD
$BWDSTART = FALSE
LDAT_ACT = LCPDAT3047
FDAT_ACT = FP3047
BAS(#CP_PARAMS, 2.0)
SET_CD_PARAMS (0)
LIN XP3047
;ENDFOLD

;FOLD LIN P3048 Vel=2 m/s CPDAT3048 Tool[1]:marker Base[0] ;%{PE}
;FOLD Parameters ;%{h}
;Params IlfProvider=kukaroboter.basistech.inlineforms.movement.old; Kuka.IsGlobalPoint=False; Kuka.PointName=P3048; Kuka.BlendingEnabled=False; Kuka.MoveDataName=CPDAT1; Kuka.VelocityPath=2; Kuka.CurrentCDSetIndex=0; Kuka.MovementParameterFieldEnabled=True; IlfCommand=LIN
;ENDFOLD
$BWDSTART = FALSE
LDAT_ACT = LCPDAT3048
FDAT_ACT = FP3048
BAS(#CP_PARAMS, 2.0)
SET_CD_PARAMS (0)
LIN XP3048
;ENDFOLD

;FOLD LIN P3049 Vel=2 m/s CPDAT3049 Tool[1]:marker Base[0] ;%{PE}
;FOLD Parameters ;%{h}
;Params IlfProvider=kukaroboter.basistech.inlineforms.movement.old; Kuka.IsGlobalPoint=False; Kuka.PointName=P3049; Kuka.BlendingEnabled=False; Kuka.MoveDataName=CPDAT1; Kuka.VelocityPath=2; Kuka.CurrentCDSetIndex=0; Kuka.MovementParameterFieldEnabled=True; IlfCommand=LIN
;ENDFOLD
$BWDSTART = FALSE
LDAT_ACT = LCPDAT3049
FDAT_ACT = FP3049
BAS(#CP_PARAMS, 2.0)
SET_CD_PARAMS (0)
LIN XP3049
;ENDFOLD

;FOLD LIN P3050 Vel=2 m/s CPDAT3050 Tool[1]:marker Base[0] ;%{PE}
;FOLD Parameters ;%{h}
;Params IlfProvider=kukaroboter.basistech.inlineforms.movement.old; Kuka.IsGlobalPoint=False; Kuka.PointName=P3050; Kuka.BlendingEnabled=False; Kuka.MoveDataName=CPDAT1; Kuka.VelocityPath=2; Kuka.CurrentCDSetIndex=0; Kuka.MovementParameterFieldEnabled=True; IlfCommand=LIN
;ENDFOLD
$BWDSTART = FALSE
LDAT_ACT = LCPDAT3050
FDAT_ACT = FP3050
BAS(#CP_PARAMS, 2.0)
SET_CD_PARAMS (0)
LIN XP3050
;ENDFOLD

;FOLD LIN P3051 Vel=2 m/s CPDAT3051 Tool[1]:marker Base[0] ;%{PE}
;FOLD Parameters ;%{h}
;Params IlfProvider=kukaroboter.basistech.inlineforms.movement.old; Kuka.IsGlobalPoint=False; Kuka.PointName=P3051; Kuka.BlendingEnabled=False; Kuka.MoveDataName=CPDAT1; Kuka.VelocityPath=2; Kuka.CurrentCDSetIndex=0; Kuka.MovementParameterFieldEnabled=True; IlfCommand=LIN
;ENDFOLD
$BWDSTART = FALSE
LDAT_ACT = LCPDAT3051
FDAT_ACT = FP3051
BAS(#CP_PARAMS, 2.0)
SET_CD_PARAMS (0)
LIN XP3051
;ENDFOLD

;FOLD LIN P3052 Vel=2 m/s CPDAT3052 Tool[1]:marker Base[0] ;%{PE}
;FOLD Parameters ;%{h}
;Params IlfProvider=kukaroboter.basistech.inlineforms.movement.old; Kuka.IsGlobalPoint=False; Kuka.PointName=P3052; Kuka.BlendingEnabled=False; Kuka.MoveDataName=CPDAT1; Kuka.VelocityPath=2; Kuka.CurrentCDSetIndex=0; Kuka.MovementParameterFieldEnabled=True; IlfCommand=LIN
;ENDFOLD
$BWDSTART = FALSE
LDAT_ACT = LCPDAT3052
FDAT_ACT = FP3052
BAS(#CP_PARAMS, 2.0)
SET_CD_PARAMS (0)
LIN XP3052
;ENDFOLD

;FOLD LIN P3053 Vel=2 m/s CPDAT3053 Tool[1]:marker Base[0] ;%{PE}
;FOLD Parameters ;%{h}
;Params IlfProvider=kukaroboter.basistech.inlineforms.movement.old; Kuka.IsGlobalPoint=False; Kuka.PointName=P3053; Kuka.BlendingEnabled=False; Kuka.MoveDataName=CPDAT1; Kuka.VelocityPath=2; Kuka.CurrentCDSetIndex=0; Kuka.MovementParameterFieldEnabled=True; IlfCommand=LIN
;ENDFOLD
$BWDSTART = FALSE
LDAT_ACT = LCPDAT3053
FDAT_ACT = FP3053
BAS(#CP_PARAMS, 2.0)
SET_CD_PARAMS (0)
LIN XP3053
;ENDFOLD

;FOLD LIN P3054 Vel=2 m/s CPDAT3054 Tool[1]:marker Base[0] ;%{PE}
;FOLD Parameters ;%{h}
;Params IlfProvider=kukaroboter.basistech.inlineforms.movement.old; Kuka.IsGlobalPoint=False; Kuka.PointName=P3054; Kuka.BlendingEnabled=False; Kuka.MoveDataName=CPDAT1; Kuka.VelocityPath=2; Kuka.CurrentCDSetIndex=0; Kuka.MovementParameterFieldEnabled=True; IlfCommand=LIN
;ENDFOLD
$BWDSTART = FALSE
LDAT_ACT = LCPDAT3054
FDAT_ACT = FP3054
BAS(#CP_PARAMS, 2.0)
SET_CD_PARAMS (0)
LIN XP3054
;ENDFOLD

;FOLD LIN P3055 Vel=2 m/s CPDAT3055 Tool[1]:marker Base[0] ;%{PE}
;FOLD Parameters ;%{h}
;Params IlfProvider=kukaroboter.basistech.inlineforms.movement.old; Kuka.IsGlobalPoint=False; Kuka.PointName=P3055; Kuka.BlendingEnabled=False; Kuka.MoveDataName=CPDAT1; Kuka.VelocityPath=2; Kuka.CurrentCDSetIndex=0; Kuka.MovementParameterFieldEnabled=True; IlfCommand=LIN
;ENDFOLD
$BWDSTART = FALSE
LDAT_ACT = LCPDAT3055
FDAT_ACT = FP3055
BAS(#CP_PARAMS, 2.0)
SET_CD_PARAMS (0)
LIN XP3055
;ENDFOLD

;FOLD LIN P3056 Vel=2 m/s CPDAT3056 Tool[1]:marker Base[0] ;%{PE}
;FOLD Parameters ;%{h}
;Params IlfProvider=kukaroboter.basistech.inlineforms.movement.old; Kuka.IsGlobalPoint=False; Kuka.PointName=P3056; Kuka.BlendingEnabled=False; Kuka.MoveDataName=CPDAT1; Kuka.VelocityPath=2; Kuka.CurrentCDSetIndex=0; Kuka.MovementParameterFieldEnabled=True; IlfCommand=LIN
;ENDFOLD
$BWDSTART = FALSE
LDAT_ACT = LCPDAT3056
FDAT_ACT = FP3056
BAS(#CP_PARAMS, 2.0)
SET_CD_PARAMS (0)
LIN XP3056
;ENDFOLD

;FOLD LIN P3057 Vel=2 m/s CPDAT3057 Tool[1]:marker Base[0] ;%{PE}
;FOLD Parameters ;%{h}
;Params IlfProvider=kukaroboter.basistech.inlineforms.movement.old; Kuka.IsGlobalPoint=False; Kuka.PointName=P3057; Kuka.BlendingEnabled=False; Kuka.MoveDataName=CPDAT1; Kuka.VelocityPath=2; Kuka.CurrentCDSetIndex=0; Kuka.MovementParameterFieldEnabled=True; IlfCommand=LIN
;ENDFOLD
$BWDSTART = FALSE
LDAT_ACT = LCPDAT3057
FDAT_ACT = FP3057
BAS(#CP_PARAMS, 2.0)
SET_CD_PARAMS (0)
LIN XP3057
;ENDFOLD

;FOLD LIN P3058 Vel=2 m/s CPDAT3058 Tool[1]:marker Base[0] ;%{PE}
;FOLD Parameters ;%{h}
;Params IlfProvider=kukaroboter.basistech.inlineforms.movement.old; Kuka.IsGlobalPoint=False; Kuka.PointName=P3058; Kuka.BlendingEnabled=False; Kuka.MoveDataName=CPDAT1; Kuka.VelocityPath=2; Kuka.CurrentCDSetIndex=0; Kuka.MovementParameterFieldEnabled=True; IlfCommand=LIN
;ENDFOLD
$BWDSTART = FALSE
LDAT_ACT = LCPDAT3058
FDAT_ACT = FP3058
BAS(#CP_PARAMS, 2.0)
SET_CD_PARAMS (0)
LIN XP3058
;ENDFOLD

;FOLD LIN P3059 Vel=2 m/s CPDAT3059 Tool[1]:marker Base[0] ;%{PE}
;FOLD Parameters ;%{h}
;Params IlfProvider=kukaroboter.basistech.inlineforms.movement.old; Kuka.IsGlobalPoint=False; Kuka.PointName=P3059; Kuka.BlendingEnabled=False; Kuka.MoveDataName=CPDAT1; Kuka.VelocityPath=2; Kuka.CurrentCDSetIndex=0; Kuka.MovementParameterFieldEnabled=True; IlfCommand=LIN
;ENDFOLD
$BWDSTART = FALSE
LDAT_ACT = LCPDAT3059
FDAT_ACT = FP3059
BAS(#CP_PARAMS, 2.0)
SET_CD_PARAMS (0)
LIN XP3059
;ENDFOLD

;FOLD LIN P3060 Vel=2 m/s CPDAT3060 Tool[1]:marker Base[0] ;%{PE}
;FOLD Parameters ;%{h}
;Params IlfProvider=kukaroboter.basistech.inlineforms.movement.old; Kuka.IsGlobalPoint=False; Kuka.PointName=P3060; Kuka.BlendingEnabled=False; Kuka.MoveDataName=CPDAT1; Kuka.VelocityPath=2; Kuka.CurrentCDSetIndex=0; Kuka.MovementParameterFieldEnabled=True; IlfCommand=LIN
;ENDFOLD
$BWDSTART = FALSE
LDAT_ACT = LCPDAT3060
FDAT_ACT = FP3060
BAS(#CP_PARAMS, 2.0)
SET_CD_PARAMS (0)
LIN XP3060
;ENDFOLD

;FOLD LIN P3061 Vel=2 m/s CPDAT3061 Tool[1]:marker Base[0] ;%{PE}
;FOLD Parameters ;%{h}
;Params IlfProvider=kukaroboter.basistech.inlineforms.movement.old; Kuka.IsGlobalPoint=False; Kuka.PointName=P3061; Kuka.BlendingEnabled=False; Kuka.MoveDataName=CPDAT1; Kuka.VelocityPath=2; Kuka.CurrentCDSetIndex=0; Kuka.MovementParameterFieldEnabled=True; IlfCommand=LIN
;ENDFOLD
$BWDSTART = FALSE
LDAT_ACT = LCPDAT3061
FDAT_ACT = FP3061
BAS(#CP_PARAMS, 2.0)
SET_CD_PARAMS (0)
LIN XP3061
;ENDFOLD

;FOLD LIN P3062 Vel=2 m/s CPDAT3062 Tool[1]:marker Base[0] ;%{PE}
;FOLD Parameters ;%{h}
;Params IlfProvider=kukaroboter.basistech.inlineforms.movement.old; Kuka.IsGlobalPoint=False; Kuka.PointName=P3062; Kuka.BlendingEnabled=False; Kuka.MoveDataName=CPDAT1; Kuka.VelocityPath=2; Kuka.CurrentCDSetIndex=0; Kuka.MovementParameterFieldEnabled=True; IlfCommand=LIN
;ENDFOLD
$BWDSTART = FALSE
LDAT_ACT = LCPDAT3062
FDAT_ACT = FP3062
BAS(#CP_PARAMS, 2.0)
SET_CD_PARAMS (0)
LIN XP3062
;ENDFOLD

;FOLD LIN P3063 Vel=2 m/s CPDAT3063 Tool[1]:marker Base[0] ;%{PE}
;FOLD Parameters ;%{h}
;Params IlfProvider=kukaroboter.basistech.inlineforms.movement.old; Kuka.IsGlobalPoint=False; Kuka.PointName=P3063; Kuka.BlendingEnabled=False; Kuka.MoveDataName=CPDAT1; Kuka.VelocityPath=2; Kuka.CurrentCDSetIndex=0; Kuka.MovementParameterFieldEnabled=True; IlfCommand=LIN
;ENDFOLD
$BWDSTART = FALSE
LDAT_ACT = LCPDAT3063
FDAT_ACT = FP3063
BAS(#CP_PARAMS, 2.0)
SET_CD_PARAMS (0)
LIN XP3063
;ENDFOLD

;FOLD LIN P3064 Vel=2 m/s CPDAT3064 Tool[1]:marker Base[0] ;%{PE}
;FOLD Parameters ;%{h}
;Params IlfProvider=kukaroboter.basistech.inlineforms.movement.old; Kuka.IsGlobalPoint=False; Kuka.PointName=P3064; Kuka.BlendingEnabled=False; Kuka.MoveDataName=CPDAT1; Kuka.VelocityPath=2; Kuka.CurrentCDSetIndex=0; Kuka.MovementParameterFieldEnabled=True; IlfCommand=LIN
;ENDFOLD
$BWDSTART = FALSE
LDAT_ACT = LCPDAT3064
FDAT_ACT = FP3064
BAS(#CP_PARAMS, 2.0)
SET_CD_PARAMS (0)
LIN XP3064
;ENDFOLD

;FOLD LIN P3065 Vel=2 m/s CPDAT3065 Tool[1]:marker Base[0] ;%{PE}
;FOLD Parameters ;%{h}
;Params IlfProvider=kukaroboter.basistech.inlineforms.movement.old; Kuka.IsGlobalPoint=False; Kuka.PointName=P3065; Kuka.BlendingEnabled=False; Kuka.MoveDataName=CPDAT1; Kuka.VelocityPath=2; Kuka.CurrentCDSetIndex=0; Kuka.MovementParameterFieldEnabled=True; IlfCommand=LIN
;ENDFOLD
$BWDSTART = FALSE
LDAT_ACT = LCPDAT3065
FDAT_ACT = FP3065
BAS(#CP_PARAMS, 2.0)
SET_CD_PARAMS (0)
LIN XP3065
;ENDFOLD

;FOLD LIN P3066 Vel=2 m/s CPDAT3066 Tool[1]:marker Base[0] ;%{PE}
;FOLD Parameters ;%{h}
;Params IlfProvider=kukaroboter.basistech.inlineforms.movement.old; Kuka.IsGlobalPoint=False; Kuka.PointName=P3066; Kuka.BlendingEnabled=False; Kuka.MoveDataName=CPDAT1; Kuka.VelocityPath=2; Kuka.CurrentCDSetIndex=0; Kuka.MovementParameterFieldEnabled=True; IlfCommand=LIN
;ENDFOLD
$BWDSTART = FALSE
LDAT_ACT = LCPDAT3066
FDAT_ACT = FP3066
BAS(#CP_PARAMS, 2.0)
SET_CD_PARAMS (0)
LIN XP3066
;ENDFOLD

;FOLD LIN P3067 Vel=2 m/s CPDAT3067 Tool[1]:marker Base[0] ;%{PE}
;FOLD Parameters ;%{h}
;Params IlfProvider=kukaroboter.basistech.inlineforms.movement.old; Kuka.IsGlobalPoint=False; Kuka.PointName=P3067; Kuka.BlendingEnabled=False; Kuka.MoveDataName=CPDAT1; Kuka.VelocityPath=2; Kuka.CurrentCDSetIndex=0; Kuka.MovementParameterFieldEnabled=True; IlfCommand=LIN
;ENDFOLD
$BWDSTART = FALSE
LDAT_ACT = LCPDAT3067
FDAT_ACT = FP3067
BAS(#CP_PARAMS, 2.0)
SET_CD_PARAMS (0)
LIN XP3067
;ENDFOLD

;FOLD LIN P3068 Vel=2 m/s CPDAT3068 Tool[1]:marker Base[0] ;%{PE}
;FOLD Parameters ;%{h}
;Params IlfProvider=kukaroboter.basistech.inlineforms.movement.old; Kuka.IsGlobalPoint=False; Kuka.PointName=P3068; Kuka.BlendingEnabled=False; Kuka.MoveDataName=CPDAT1; Kuka.VelocityPath=2; Kuka.CurrentCDSetIndex=0; Kuka.MovementParameterFieldEnabled=True; IlfCommand=LIN
;ENDFOLD
$BWDSTART = FALSE
LDAT_ACT = LCPDAT3068
FDAT_ACT = FP3068
BAS(#CP_PARAMS, 2.0)
SET_CD_PARAMS (0)
LIN XP3068
;ENDFOLD

;FOLD LIN P3069 Vel=2 m/s CPDAT3069 Tool[1]:marker Base[0] ;%{PE}
;FOLD Parameters ;%{h}
;Params IlfProvider=kukaroboter.basistech.inlineforms.movement.old; Kuka.IsGlobalPoint=False; Kuka.PointName=P3069; Kuka.BlendingEnabled=False; Kuka.MoveDataName=CPDAT1; Kuka.VelocityPath=2; Kuka.CurrentCDSetIndex=0; Kuka.MovementParameterFieldEnabled=True; IlfCommand=LIN
;ENDFOLD
$BWDSTART = FALSE
LDAT_ACT = LCPDAT3069
FDAT_ACT = FP3069
BAS(#CP_PARAMS, 2.0)
SET_CD_PARAMS (0)
LIN XP3069
;ENDFOLD

;FOLD LIN P3070 Vel=2 m/s CPDAT3070 Tool[1]:marker Base[0] ;%{PE}
;FOLD Parameters ;%{h}
;Params IlfProvider=kukaroboter.basistech.inlineforms.movement.old; Kuka.IsGlobalPoint=False; Kuka.PointName=P3070; Kuka.BlendingEnabled=False; Kuka.MoveDataName=CPDAT1; Kuka.VelocityPath=2; Kuka.CurrentCDSetIndex=0; Kuka.MovementParameterFieldEnabled=True; IlfCommand=LIN
;ENDFOLD
$BWDSTART = FALSE
LDAT_ACT = LCPDAT3070
FDAT_ACT = FP3070
BAS(#CP_PARAMS, 2.0)
SET_CD_PARAMS (0)
LIN XP3070
;ENDFOLD

;FOLD LIN P3071 Vel=2 m/s CPDAT3071 Tool[1]:marker Base[0] ;%{PE}
;FOLD Parameters ;%{h}
;Params IlfProvider=kukaroboter.basistech.inlineforms.movement.old; Kuka.IsGlobalPoint=False; Kuka.PointName=P3071; Kuka.BlendingEnabled=False; Kuka.MoveDataName=CPDAT1; Kuka.VelocityPath=2; Kuka.CurrentCDSetIndex=0; Kuka.MovementParameterFieldEnabled=True; IlfCommand=LIN
;ENDFOLD
$BWDSTART = FALSE
LDAT_ACT = LCPDAT3071
FDAT_ACT = FP3071
BAS(#CP_PARAMS, 2.0)
SET_CD_PARAMS (0)
LIN XP3071
;ENDFOLD

;FOLD LIN P3072 Vel=2 m/s CPDAT3072 Tool[1]:marker Base[0] ;%{PE}
;FOLD Parameters ;%{h}
;Params IlfProvider=kukaroboter.basistech.inlineforms.movement.old; Kuka.IsGlobalPoint=False; Kuka.PointName=P3072; Kuka.BlendingEnabled=False; Kuka.MoveDataName=CPDAT1; Kuka.VelocityPath=2; Kuka.CurrentCDSetIndex=0; Kuka.MovementParameterFieldEnabled=True; IlfCommand=LIN
;ENDFOLD
$BWDSTART = FALSE
LDAT_ACT = LCPDAT3072
FDAT_ACT = FP3072
BAS(#CP_PARAMS, 2.0)
SET_CD_PARAMS (0)
LIN XP3072
;ENDFOLD

